(* CODESYS project RoboConnect_Dobot.library
   Company: RoboConnect
   DefaultNamespace: RoboConnect.Dobot
   Version: 0.1.0.0
   Placeholder: RoboConnect.Dobot
   Author: RoboConnect_Maintainers
   Description: 0.1.0.0 Branding update
      
      0.0.11.0 corrected MovJ arrays with checks
      0.0.10.0 adds free all tasks
      0.0.9.x - WIP
      0.0.9.0 refactors command creator
      0.0.8.0 updates to new Param name in TcRobot lib
      0.0.7.0 using new command infrastructure 
      0.0.0.6 command task receives 
      0.0.0.5 - updating array sizes
      0.0.0.3 adding receive packet scanning.
      0.0.0.2  adding separate port classes.
      0.0.0.1 Initial
   Title: RoboConnect.Dobot

Project tree, tasks and I/O mapping:
  libraries: Intecre.Utilities, * (Intecre Ltd); RoboConnect, * (RoboConnect); Tc2_Standard, * (Beckhoff Automation GmbH); Tc2_System, * (Beckhoff Automation GmbH); Tc2_Utilities, * (Beckhoff Automation GmbH)
  Commands and tasks/
    function block T_BoolCommandTaskV3 [ST]: Result, SetResultValue
    function block T_CommandTaskPoolV3 [ST]: FreeAllTasks, GetTask
    function block T_CommandTaskV3 [ST]: Abort, CyclicLogic, Execute, Free, Initalise, StateChanged, Available, Busy, Done, Error, ErrorId, Timeout
    function block T_DobotCommandConstructor [ST]: BrakeControl, ClearError, ContinueImmediate, ContinueScript, DisableRobot, EmergencyStop, EnableRobot, EnableRobotSpecifyCoG, Pause, PauseScript, PowerOn, ResetRobot, RunScript, SetCollideDrag, SetSafeSkin, StartDrag, StopDrag, StopScript, Wait, AccJ, AccL, CalcTool, CalcUser, Cp, LoadSwitch, PayLoad, SetArmOrientation, SetCollisionLevel, SetTool, SetUser, SpeedFactor, SpeedJ, SpeedL, TcpSpeed, TcpSpeedEnd, Tool, User, GetAngle, GetErrorID, GetPalletPose, GetPathStartPose, GetPose, GetSixForceData, GetTraceStartPose, HandleTrajPoints, InverseSolution, PalletCreate, PositiveSolution, RobotMode, AnalogueInput, AnalogueOutput, AoExecute, DigitalInput, DigitalOutput, DiGroup, DoExecute, DoGroup, GetTerminal485, SetTerminal485, ToolAI, ToolDI, ToolDO, ToolDOExecute, GetCoils, GetHoldRegs, GetInBits, GetInRegs, ModbusClose, ModbusCreate, SetCoils, SetHoldRegs, Circle3, Circle3Advanced, MoveJogCartesian, MoveJogCartesianAdvanced, MoveJogJointAxis, MoveJogJointAxisAdvanced, JointMovJ, JointMovJAdvanced, MovJ, MovJAdvanced, MovJIO, MovJIOAdvanced, MovL, MovLAdvanced, MovLIO, MovLIOAdvanced, RelJointMovJ, RelJointMovJAdvanced, RelMovJTool, RelMovJToolAdvanced, RelMovJUser, RelMovJUserAdvanced, RelMovLTool, RelMovLToolAdvanced, RelMovLUser, RelMovLUserAdvanced, ServoJ, ServoJAdvanced, Arc, ServoP, StartPath, StartTrace, Sync, CreateCommand, CreateCommand_EightArgs, CreateCommand_ElevenArgs, CreateCommand_Fifteen_Args, CreateCommand_FiveArgs, CreateCommand_FourArgs, CreateCommand_NineArgs, CreateCommand_OneArg, CreateCommand_SevenArgs, CreateCommand_SixArgs, CreateCommand_TenArgs, CreateCommand_Thirteen_Args, CreateCommand_ThreeArgs, CreateCommand_TwoArgs, CreateCommandNoArgs, EncapsulateWithCurlyBrax
    function block T_NumberCommandTaskV3 [ST]: Result, SetResultValue
  Helpers/
    function arrayToString [ST]
    function ByteArrayAdvanceAndClearRemaining [ST]
    function F_GetNextSegmentAndRemove [ST]
    function F_RemoveAfterSemiColon [ST]
    function F_RemoveAllOfACharacterInPlace [ST]
  Project Information/
    function F_GetCompany [ST]
    function F_GetTitle [ST]
    function F_GetVersion [ST]
  Structs and Enums/
    data type Converter2Bytes
    data type Converter8Bytes
    data type DOBOT_CMD_STRING
    data type DobotCR3Feedback
    data type E_BrakeControlRequest
    data type E_DobotTypes
    data type RobotModeConverter
    data type RobotModes
    data type TargetJogCrNova
  V3_API/
    function block T_DashboardV3 [ST]: ClearError, Disable, Enable, Halt, Reset, Stop, SetAnalogOutput, SetBufferMode, SetCarteasianAcceleration, SetCartesianDynamics, SetCartesianSpeed, SetDigitalOutput, SetJointAcceleration, SetJointSpeed, SetToolAnalogOutput, SetToolDigitalOutput, SetToolFrame, SetTransitionMode, SetTransitionParameter, SetUserFrame, ClearQueue, Connect, Disconnect, FreeAllTasks, SetRobotType, CallRobotApi, CallRobotApi_NormalPriority, Connected, DobotType
    function block T_FeedbackV3 [ST]: ClearAccumulator, Connect, CyclicReadFeedback, Disconnect, AdvanceAccumulatorArray, DecodeFeedback, Connected, Error, ErrorID, RobotFdBack
    function block T_MotionV3 [ST]: ClearQueue, Connect, Disconnect, FreeAllTasks, JogCartesian, JogJointAxis, MoveAbs, MoveJ, SetRobotType, CallRobotApi, CallRobotApi_NormalPriority, Connected, DobotType
    function block T_V3CommandAndFeedbackBaseClass [ST]: StateChanged, Connected, DobotType, CallRobotApi, ClearQueue, Connect, Disconnect, FreeAllTasks, Initialise, SetRobotType
    global variables V3_Ports
  Version/
    global variables Global_Version
  function block T_DobotV3_Cr_Nova [ST]: GetAnalogOutput, GetAxisCurrents, GetAxisPositions, GetAxisTemperatures, GetDigitalOutput, GetToolAnalogOutput, GetToolDigitalOutput, ClearError, Connect, CyclicLogic, Disable, Disconnect, Enable, FreeAllTasks, GetJointPositions, Halt, IsAtCartesianPosition, IsAtJointPosition, JogAxis, JogAxisAdvanced, JogCartesian, JogJointAxis, MoveAbs, MoveJ, Reset, SetAtPosDeltas, StateChanged, Stop, CartesianPosition, Connected, Enabled, Error, ErrorID, Manufacturer, Model, Running, ToolPosition, SetAnalogOutput, SetBufferMode, SetCarteasianAcceleration, SetCartesianDynamics, SetCartesianSpeed, SetDigitalOutput, SetJointAcceleration, SetJointSpeed, SetToolAnalogOutput, SetToolDigitalOutput, SetToolFrame, SetTransitionMode, SetTransitionParameter, SetUserFrame, FB_init, SetConnectionProperties
*)

// Structs and Enums/Converter2Bytes
TYPE Converter2Bytes :
UNION
	arrBytesIn : ARRAY[0..1] OF BYTE;
	realOut : INT;
END_UNION
END_TYPE

// Structs and Enums/Converter8Bytes
TYPE Converter8Bytes :
UNION
	arrBytesIn : ARRAY[0..7] OF BYTE;
	wordOut : LWORD;
	realOut : LREAL;
END_UNION
END_TYPE

// Structs and Enums/DOBOT_CMD_STRING
TYPE DOBOT_CMD_STRING : STRING(255); END_TYPE

// Structs and Enums/DobotCR3Feedback
TYPE DobotCR3Feedback :
STRUCT
	MessageSize : Converter2Bytes;
	DigitalInputs : ARRAY[0..8] OF BOOL;
	DigitalOutputs : ARRAY[0..8]OF BOOL;
	RobotMode : RobotModeConverter;
	TimeStamp : Converter8Bytes;
	TestValue :  Converter8Bytes;
	SpeedScaling : Converter8Bytes;
	LinearMomentumNorm : Converter8Bytes;
	VMain : Converter8Bytes;
	VRobot : Converter8Bytes;
	IRobot : Converter8Bytes;
	ToolAcceleroMeter : ARRAY[0..2] OF Converter8Bytes;
	ElbowPosition 	: ARRAY[0..2] OF Converter8Bytes;
	ElbowVelocity 	: ARRAY[0..2] OF Converter8Bytes;
	QTarget : ARRAY[0..5] OF Converter8Bytes; 	
	QDTarget : ARRAY[0..5] OF Converter8Bytes; 	
	QDDTarget : ARRAY[0..5] OF Converter8Bytes; 	
	ITarget : ARRAY[0..5] OF Converter8Bytes;	
	MTarget : ARRAY[0..5] OF Converter8Bytes;	
	QActual : ARRAY[0..5] OF Converter8Bytes;	
	QDActual : ARRAY[0..5] OF Converter8Bytes;
	IActual : ARRAY[0..5] OF Converter8Bytes;
	ActualTCPForce : ARRAY[0..5] OF Converter8Bytes;
	ToolVectorActual  : ARRAY[0..5] OF Converter8Bytes;	
	TCPSpeedActual : ARRAY[0..5] OF Converter8Bytes; 	
	TCPForce : ARRAY[0..5] OF Converter8Bytes; 	
	ToolVectorTarget : ARRAY[0..5] OF Converter8Bytes; 	
	TCPSpeedTarget : ARRAY[0..5] OF Converter8Bytes; 	
	MotorTemperatures : ARRAY[0..5] OF Converter8Bytes; 	
	JointModes : ARRAY[0..5] OF Converter8Bytes; 
	VActual : ARRAY[0..5] OF Converter8Bytes; 	
	HandType : ARRAY[0..3] OF BYTE; 	
	User : BYTE; 	
	Tool: Converter2Bytes;  	
	RunQueuedCmd: BOOL;  	
	PauseCmdFlag : BOOL; 	
	VelocityRatio: REAL;  	
	AccelerationRatio : REAL; 	
	JerkRatio 	: REAL; 
	XYZVelocityRatio: REAL;  	
	RVelocityRatio: REAL;  
	XYZAccelerationRatio: REAL;  	
	RAccelerationRatio : REAL; 	
	XYZJerkRatio : REAL; 	
	RJerkRatio : REAL; 	
	BrakeStatus : BOOL; 	
	EnableStatus : BOOL; 	
	DragStatus : BOOL; 	
	RunningStatus : BOOL; 	
	ErrorStatus : BOOL; 	
	JogStatusCR 	: BOOL; 
	CRRobotType : INT; 	
	DragButtonSignal : BOOL; 	
	EnableButtonSignal : BOOL; 	
	RecordButtonSignal : BOOL; 
	ReappearButtonSignal : BOOL; 	
	JawButtonSignal  : BOOL; 	
	SixForceOnline : BOOL; 	
	MActual : ARRAY[0..5] OF Converter8Bytes; 	 
	Load : ARRAY[0..4] OF REAL;  	
	CenterX : Converter2Bytes; 	
	CenterY  : Converter2Bytes;	
	CenterZ  : Converter2Bytes;	
//	User  : ARRAY[0..5] OF Converter8Bytes; 	 	
	ToolCordinates  : ARRAY[0..5] OF Converter8Bytes; 	 	
	TraceIndex : Converter8Bytes; 	
	SixForceValue  : ARRAY[0..5] OF Converter8Bytes; 		
	TargetQuaternion  : ARRAY[0..3] OF Converter8Bytes; 		
	ActualQuaternion : ARRAY[0..3] OF Converter8Bytes; 	
END_STRUCT
END_TYPE

// Structs and Enums/E_BrakeControlRequest
{attribute 'qualified_only'}
{attribute 'strict'}
TYPE E_BrakeControlRequest :
(
	NONE,
  ON,
  OFF
);
END_TYPE

// Structs and Enums/E_DobotTypes
{attribute 'qualified_only'}
{attribute 'to_string'}
{attribute 'strict'}
TYPE
E_DobotTypes :
(
  NONE,
  CR3, // 6 dof
  CR5, // 6 dof
  CR7, // 6 dof
  CR10, // 6 dof
  CR12, // 6 dof
  CR16, // 6 dof
  NOVA_2, // 6 dof
  NOVA_5, // 6 dof
  MG400 // 4 dof
);
END_TYPE

// Structs and Enums/RobotModeConverter
TYPE RobotModeConverter :
UNION
	arrBytesIn : ARRAY[0..7] OF BYTE;
	robotMode : INT;
END_UNION
END_TYPE

// Structs and Enums/RobotModes
{attribute 'qualified_only'}
{attribute 'to_string'}
TYPE
RobotModes :
(
  Not_Connected := 0,
  Initialization := 1,
  Brake_Release := 2,
  Disable := 4,
  Enable := 5,
  Dragging_State := 6,
  Running_State := 7,
  Draggin_Recording := 8,
  Alarm_State := 9,
  Pause_State := 10,
  Jogging_State := 11
) INT;
END_TYPE

// Structs and Enums/TargetJogCrNova
TYPE TargetJogCrNova :
(
	StopJog := 0,
	x := 1,
	y := 2,
	z := 3,
	a := 4,
	b := 5,
	c := 6	
);
END_TYPE

// V3_API/V3_Ports
{attribute 'qualified_only'}
VAR_GLOBAL CONSTANT
  FEEDBACK : UINT := 30004;
  DASHBOARD : UINT := 29999;
  MOTION : UINT := 30003;
END_VAR

// Version/Global_Version
{attribute 'TcGenerated'}
{attribute 'no-analysis'}
{attribute 'linkalways'}
// This function has been automatically generated from the project information.
VAR_GLOBAL CONSTANT
	{attribute 'const_non_replaced'}
	stLibVersion_RoboConnect_Dobot : ST_LibVersion := (iMajor := 0, iMinor := 1, iBuild := 0, iRevision := 0, nFlags := 0, sVersion := '0.1.0.0');
END_VAR

// Commands and tasks/T_BoolCommandTaskV3
FUNCTION_BLOCK T_BoolCommandTaskV3 EXTENDS T_CommandTaskV3 IMPLEMENTS I_BoolResultTask
VAR
  _boolResult : BOOL;
END_VAR

PROPERTY Result : BOOL
GET
Result := _boolResult;
END_GET
END_PROPERTY

METHOD PUBLIC SetResultValue
VAR_INPUT
  value : BOOL;
END_VAR
_boolResult := value;
END_METHOD

END_FUNCTION_BLOCK

// Commands and tasks/T_CommandTaskV3
FUNCTION_BLOCK T_CommandTaskV3 EXTENDS T_NamedBase IMPLEMENTS I_CommandTask
VAR
  _busy : BOOL := FALSE;
  _error : BOOL := FALSE;
  _done : BOOL := FALSE;
  _errorId : STRING;
  _result : DOBOT_CMD_STRING;
  _timeout : BOOL := FALSE;
  _available : BOOL := TRUE;

  state, prevState : (UNINITLIASED,
    INITALISED,
    SENDING,
    WAITING_FOR_RESPONSE,
    DONE_STATE,
    ERROR_STATE);

  _comPort : I_Connection;
  _msg : T_Maxstring;
  
  timeoutTimer : TON := (PT := TASK_TIMEOUT);
  data : RecvBuffer;
  receiveLength : UDINT;
  resultString : DOBOT_CMD_STRING;
  origRequestPosition : INT;
  errorString : T_Maxstring;
  originalReq : DOBOT_CMD_STRING;
  errorCode : DOBOT_CMD_STRING;
  results : DOBOT_CMD_STRING;
  spaceString : STRING := ' ';
  tempResString : DOBOT_CMD_STRING;

END_VAR
VAR CONSTANT
  TASK_TIMEOUT : TIME := RoboConnect.RoboConnectParams.TimeOut;
END_VAR

METHOD Abort
END_METHOD

METHOD PUBLIC CyclicLogic
CASE state OF
  UNINITLIASED:
    StateChanged();

  INITALISED:
    IF StateChanged() THEN
      logInfo('task initlaised');
    END_IF

  SENDING:
    IF StateChanged() THEN
      _busy := TRUE;
      timeoutTimer.IN := FALSE;

      IF NOT _comPort.Send(_msg) THEN
        state := ERROR_STATE;
        RETURN;

      END_IF

    ELSE
      timeoutTimer.IN := TRUE;
    END_IF

    IF timeoutTimer.Q THEN
      state := ERROR_STATE;
      LogError('Command timed out');
    END_IF

    IF _comPort.SendDone THEN
      state := WAITING_FOR_RESPONSE;
    END_IF

  WAITING_FOR_RESPONSE:
    timeoutTimer.IN := NOT StateChanged();

    IF timeoutTimer.Q THEN
      LogError('No return from sent command!');
      state := ERROR_STATE;

    ELSIF _comPort.IsErrorConnect OR _comPort.IsErrorReceive THEN
      LogError('_comPort.IsErrorConnect OR _comPort.IsErrorReceive');
      state := ERROR_STATE;

    ELSIF _comPort.Receive(data => data, receiveLength => receiveLength) THEN
      // convert to string
      MEMCPY(ADR(resultString), ADR(data), receiveLength);

      // Break up parts of the command
      errorCode := F_GetNextSegmentAndRemove(resultString, ',');
      results := F_GetNextSegmentAndRemove(resultString, ',');
      originalReq := F_RemoveAfterSemiColon(resultString);
      F_RemoveAllOfACharacterInPlace(original := originalReq, stringToRemove := spaceString );

      // Check what was send is what was received 
      IF originalReq = _msg THEN
        _errorId := errorCode;
        _error := errorCode <> TO_STRING(0);
        _result := results;
        state := DONE_STATE;

      ELSE
        LogError(CONCAT('Response does not contain request:', originalReq));
        LogError(CONCAT('Original request:', _msg));
        state := ERROR_STATE;

      END_IF
    END_IF

  DONE_STATE:
    IF StateChanged() THEN
      LogInfo('task done');
      _busy := FALSE;
      _done := TRUE;
      timeoutTimer.IN := FALSE;
    END_IF

  ERROR_STATE:
    IF StateChanged() THEN
      LogError('task error');
      _error := TRUE;
      _busy := FALSE;
      _done := FALSE;
    END_IF

END_CASE

timeoutTimer();
END_METHOD

METHOD PUBLIC Execute : BOOL
IF state <> INITALISED THEN
  RETURN;
END_IF

state := SENDING;
Execute := TRUE;
END_METHOD

METHOD PUBLIC Free
_Busy := FALSE;
_Error := FALSE;
_Done := FALSE;
 _timeout := FALSE;
 _available := TRUE;
  
_comPort := 0;
_msg := '';
END_METHOD

METHOD PUBLIC Initalise : BOOL
VAR_INPUT
 comPort : I_Connection;
 msg : T_Maxstring;
END_VAR
IF comPort = 0 THEN
  RETURN;
END_IF

_done := FALSE;
_comPort := comPort;
_msg := msg;
state := INITALISED;
Initalise := TRUE;
_available := false;
END_METHOD

METHOD PRIVATE StateChanged : BOOL
IF  state = prevState THEN
  RETURN;
END_IF

prevState := state;
StateChanged := TRUE;
END_METHOD

PROPERTY Available : BOOL
GET
Available := _available;
END_GET
END_PROPERTY

PROPERTY Busy : BOOL
GET
Busy := _Busy;
END_GET
END_PROPERTY

PROPERTY Done : BOOL
GET
Done := _Done;
END_GET
END_PROPERTY

PROPERTY Error : BOOL
GET
Error := _error;
END_GET
END_PROPERTY

PROPERTY PUBLIC ErrorId : STRING
GET
ErrorId := _errorId;
END_GET
END_PROPERTY

PROPERTY Timeout : BOOL
GET
Timeout := _timeout;
END_GET
END_PROPERTY

END_FUNCTION_BLOCK

// Helpers/F_GetNextSegmentAndRemove
FUNCTION INTERNAL F_GetNextSegmentAndRemove : STRING // returned segment. Does not include split character
VAR_IN_OUT
	OriginalString : STRING; // this string will be modified if split character found.
END_VAR
VAR_INPUT
	CharacterToSplitOn : STRING; // first character of this string shall be used	
END_VAR

IF LEN( OriginalString ) > 0 AND_THEN LEN( CharacterToSplitOn ) > 0 THEN

	F_GetNextSegmentAndRemove := 
		LEFT( 
			OriginalString, 
			FIND( OriginalString, LEFT( CharacterToSplitOn, 1 ) ) - 1 // do not retun the splitting character
		);
		
	OriginalString := 
		DELETE(
			OriginalString, 
			FIND( OriginalString, LEFT( CharacterToSplitOn, 1 ) ), 
			1 
		);
		
END_IF

END_FUNCTION

// Helpers/F_RemoveAfterSemiColon
FUNCTION F_RemoveAfterSemiColon : STRING
VAR_IN_OUT
  OriginalString : STRING;
END_VAR
VAR
  semiColonIndex : INT;
  semiColon : STRING := ';';
END_VAR

IF LEN(OriginalString) > 1 THEN
  semiColonIndex := FIND(OriginalString, semiColon);
  OriginalString := LEFT(OriginalString, semiColonIndex - 1);
  F_RemoveAfterSemiColon := LEFT(OriginalString, semiColonIndex - 1);
END_IF

END_FUNCTION

// Helpers/F_RemoveAllOfACharacterInPlace
FUNCTION F_RemoveAllOfACharacterInPlace 
VAR_IN_OUT
  original : DOBOT_CMD_STRING;
END_VAR
VAR_INPUT
  stringToRemove : STRING;
END_VAR
VAR
  _stringToRemove : STRING := ' ';
  tempResString : DOBOT_CMD_STRING;
END_VAR

_stringToRemove := stringToRemove;

WHILE FindAndDelete(
  pSrcString := ADR(original),
  pDeleteString := ADR(_stringToRemove),
  pDstString := ADR(tempResString),
  nDstSize := SIZEOF(tempResString)
      )
        > 0 DO

  // put back in to recursively remove spaces
  original := tempResString;

END_WHILE

END_FUNCTION

// Commands and tasks/T_CommandTaskPoolV3
FUNCTION_BLOCK T_CommandTaskPoolV3 IMPLEMENTS I_TaskPool
VAR
  taskList : ARRAY [0..MAX_TASK_SIZE] OF T_CommandTaskV3;
END_VAR
VAR CONSTANT
  MAX_TASK_SIZE : UINT := 56;
END_VAR

METHOD PUBLIC FreeAllTasks
VAR
  i : UINT;
END_VAR
FOR i := 0 TO MAX_TASK_SIZE DO
  taskList[i].Free();
END_FOR
END_METHOD

METHOD PUBLIC GetTask : BOOL
VAR_OUTPUT
  result : I_CommandTask;
END_VAR
VAR
  i : UINT;
END_VAR
FOR i := 0 TO MAX_TASK_SIZE DO
  IF taskList[i].Available THEN
    result := taskList[i];
    GetTask := TRUE;
    RETURN;
  END_IF
END_FOR

GetTask := FALSE;
END_METHOD

END_FUNCTION_BLOCK

// Commands and tasks/T_DobotCommandConstructor
FUNCTION_BLOCK T_DobotCommandConstructor EXTENDS T_NamedBase

METHOD BrakeControl : BOOL
VAR_INPUT
	axisID : INT; //joint ID, 1: J1, 2: J2, and so on
	brakeRequest : E_BrakeControlRequest; 
END_VAR
VAR_OUTPUT
	commandOutput : DOBOT_CMD_STRING;
END_VAR
VAR
  translatedBrakeValue : INT; // from Doboot API 0: Switch off brake, 1: Switch on brake
END_VAR
VAR CONSTANT
  BRAKE_CONTROL_CMD : STRING := 'BrakeControl';
END_VAR
CASE brakeRequest OF

  E_BrakeControlRequest.ON:
    translatedBrakeValue := 1;

  E_BrakeControlRequest.OFF:
    translatedBrakeValue := 0;

ELSE

  LogWarning('Cannot request Brake Control as brakeRequest = E_BrakeControlRequest.NONE ');
  RETURN;

END_CASE

commandOutput := CreateCommand_TwoArgs(BRAKE_CONTROL_CMD, TO_STRING(axisID), TO_STRING(translatedBrakeValue));

BrakeControl := TRUE;
END_METHOD

METHOD ClearError : BOOL
VAR_OUTPUT
	commandOutput : DOBOT_CMD_STRING;
END_VAR
VAR CONSTANT
	CLEAR_ERROR_CMD : STRING := 'ClearError';
END_VAR
commandOutput := CreateCommandNoArgs(CLEAR_ERROR_CMD);
ClearError := TRUE;
END_METHOD

METHOD ContinueImmediate : BOOL
VAR_OUTPUT
	commandOutput : DOBOT_CMD_STRING;
END_VAR
VAR CONSTANT
	CONTINUE_IMMEDIATE_CMD : STRING := 'Continue';
END_VAR
commandOutput := CreateCommandNoArgs(CONTINUE_IMMEDIATE_CMD);
ContinueImmediate := TRUE;
END_METHOD

METHOD ContinueScript : BOOL
VAR_OUTPUT
	commandOutput : DOBOT_CMD_STRING;
END_VAR
VAR CONSTANT
	CONTINUE_SCRIPT_CMD : STRING := 'ContinueScript';
END_VAR
commandOutput := CreateCommandNoArgs(CONTINUE_SCRIPT_CMD);
ContinueScript := TRUE;
END_METHOD

METHOD DisableRobot : BOOL
VAR_OUTPUT
	commandOutput : DOBOT_CMD_STRING;
END_VAR
VAR CONSTANT
	DISABLE_ROBOT_CMD : STRING := 'DisableRobot';
END_VAR
commandOutput := CreateCommandNoArgs(DISABLE_ROBOT_CMD);
DisableRobot := TRUE;
END_METHOD

METHOD EmergencyStop : BOOL
VAR_OUTPUT
	commandOutput : DOBOT_CMD_STRING;
END_VAR
VAR CONSTANT
	EMERGENCY_STOP_CMD : STRING := 'EmergencyStop';
END_VAR
commandOutput := CreateCommandNoArgs(EMERGENCY_STOP_CMD);
EmergencyStop := TRUE;
END_METHOD

METHOD EnableRobot : BOOL
VAR_OUTPUT
	commandOutput : DOBOT_CMD_STRING;
END_VAR
VAR CONSTANT
	ENABLE_ROBOT_CMD : DOBOT_CMD_STRING := 'EnableRobot';
END_VAR
commandOutput := CreateCommandNoArgs(ENABLE_ROBOT_CMD);
EnableRobot := TRUE;
END_METHOD

METHOD EnableRobotSpecifyCoG : BOOL // enable while specifying load and load CoG.
{attribute 'obsolete' := 'This input is optional'}
VAR_INPUT
  load : REAL := 0; //Load weight.The value range should not exceed the load range of corresponding robot models, unit: kg.
  centreX : REAL := 0; //Eccentric distance in X-axis direction. Range: -500 – 500, unit: mm.
  centreY : REAL := 0; //Eccentric distance in Y-axis direction. Range: -500 – 500, unit: mm.
  centreZ : REAL := 0; //Eccentric distance in Z-axis direction. Range: -500 – 500, unit: mm.
END_VAR
VAR_OUTPUT
  commandOutput : DOBOT_CMD_STRING;
END_VAR
VAR CONSTANT
  UPPER_LOAD_DISTANCE_BOUND : LREAL := 500; // mm
  LOWER_LOAD_DISTANCE_BOUND : LREAL := -500; // mm
  ENABLE_ROBOT_CMD : STRING := 'EnableRobot';
END_VAR
IF centreX < LOWER_LOAD_DISTANCE_BOUND OR centreX > UPPER_LOAD_DISTANCE_BOUND THEN
  LogWarning(
    CONCAT('cannot EnableRobotSpecifyCoG as centerX exceeds bounds : ', TO_STRING(centreX))
  );

  RETURN;

END_IF

IF centreY < LOWER_LOAD_DISTANCE_BOUND OR centreY > UPPER_LOAD_DISTANCE_BOUND THEN
  LogWarning(
    CONCAT('cannot EnableRobotSpecifyCoG as centreY exceeds bounds : ', TO_STRING(centreY))
  );

  RETURN;

END_IF

IF centreZ < LOWER_LOAD_DISTANCE_BOUND OR centreZ > UPPER_LOAD_DISTANCE_BOUND THEN
  LogWarning(
    CONCAT('cannot EnableRobotSpecifyCoG as centreZ exceeds bounds : ', TO_STRING(centreZ))
  );

  RETURN;

END_IF

commandOutput := CreateCommand_FourArgs(
  ENABLE_ROBOT_CMD,
  TO_STRING(load),
  TO_STRING(centreX),
  TO_STRING(centreY),
  TO_STRING(centreZ)
);

EnableRobotSpecifyCoG := TRUE;
END_METHOD

METHOD Pause : BOOL
VAR_OUTPUT
	commandOutput : DOBOT_CMD_STRING;
END_VAR
VAR CONSTANT
	PAUSE_CMD : STRING := 'Pause';
END_VAR
commandOutput := CreateCommandNoArgs(PAUSE_CMD);
Pause := TRUE;
END_METHOD

METHOD PauseScript : BOOL
VAR_OUTPUT
	commandOutput : DOBOT_CMD_STRING;
END_VAR
VAR CONSTANT
	PAUSE_SCRIPT_CMD : STRING := 'PauseScript';
END_VAR
commandOutput := CreateCommandNoArgs(PAUSE_SCRIPT_CMD);
PauseScript := TRUE;
END_METHOD

METHOD PowerOn : BOOL 
VAR_OUTPUT
	commandOutput : STRING;
END_VAR
VAR
	POWER_ON_CMD : STRING := 'PowerOn';
END_VAR
commandOutput := CreateCommandNoArgs(POWER_ON_CMD);
PowerOn := TRUE;
END_METHOD

METHOD ResetRobot : BOOL
VAR_OUTPUT
	commandOutput : DOBOT_CMD_STRING;
END_VAR
VAR CONSTANT
	RESET_ROBOT_CMD : STRING := 'ResetRobot';
END_VAR
commandOutput := CreateCommandNoArgs(RESET_ROBOT_CMD);
ResetRobot := TRUE;
END_METHOD

METHOD RunScript : BOOL
VAR_INPUT
	projectName : STRING; //Project name as created using Dobot Studio Pro
END_VAR
VAR_OUTPUT
	commandOutput : DOBOT_CMD_STRING;
END_VAR
VAR CONSTANT
	RUN_SCRIPT_CMD : STRING := 'RunScript';
END_VAR
commandOutput := CreateCommand_OneArg(RUN_SCRIPT_CMD, projectName);
RunScript := TRUE;
END_METHOD

METHOD SetCollideDrag : BOOL
VAR_INPUT
	status : INT; //Forced drag switch. 0: Forced to exit the drag mode. 1: forced to enter the drag mode.
END_VAR
VAR_OUTPUT
	commandOutput : DOBOT_CMD_STRING;
END_VAR
VAR CONSTANT
	SET_COLLIDE_DRAG_CMD : STRING := 'SetCollideDrag';
END_VAR
commandOutput := CreateCommand_OneArg(baseCommand := SET_COLLIDE_DRAG_CMD, arg_01 := TO_STRING(status));

SetCollideDrag := TRUE;
END_METHOD

METHOD SetSafeSkin : BOOL
VAR_INPUT
  status : INT; //SafeSkin switch, 0: off, 1: on
END_VAR
VAR_OUTPUT
  commandOutput : DOBOT_CMD_STRING;
END_VAR
VAR CONSTANT
  SET_SAFE_SKIN_CMD : STRING := 'SetSafeSkin';
END_VAR
commandOutput := CreateCommand_OneArg(baseCommand := SET_SAFE_SKIN_CMD, arg_01 := TO_STRING(status));

setSafeSkin := TRUE;
END_METHOD

METHOD StartDrag : BOOL
VAR_OUTPUT
	commandOutput : DOBOT_CMD_STRING;
END_VAR
VAR CONSTANT
	START_DRAG_CMD : STRING := 'StartDrag';
END_VAR
commandOutput := CreateCommandNoArgs( START_DRAG_CMD);
startDrag := TRUE;
END_METHOD

METHOD StopDrag : BOOL
VAR_OUTPUT
	commandOutput : DOBOT_CMD_STRING;
END_VAR
VAR CONSTANT
	STOP_DRAG_CMD : STRING := 'StopDrag';
END_VAR
commandOutput := CreateCommandNoArgs(STOP_DRAG_CMD);
stopDrag := TRUE;
END_METHOD

METHOD StopScript : BOOL
VAR_OUTPUT
	commandOutput : DOBOT_CMD_STRING;
END_VAR
VAR CONSTANT
	STOP_SCRIPT_CMD : DOBOT_CMD_STRING := 'StopScript';
END_VAR
commandOutput := CreateCommandNoArgs( STOP_SCRIPT_CMD);
stopScript := TRUE;
END_METHOD

METHOD Wait : BOOL
VAR_INPUT
  timeToWait : INT; //Delayed time, unit:ms, range: (0,3600*1000)
END_VAR
VAR_OUTPUT
  commandOutput : DOBOT_CMD_STRING;
END_VAR
VAR CONSTANT
  WAIT_CMD : STRING := 'Wait';
END_VAR
commandOutput := CreateCommand_OneArg(baseCommand := WAIT_CMD, arg_01 := TO_STRING(timeToWait));

Wait := TRUE;
END_METHOD

METHOD AccJ : BOOL
VAR_INPUT
	acc : INT ; //Acceleration ratio: [1-100]
END_VAR
VAR_OUTPUT
	commandOutput : DOBOT_CMD_STRING;
END_VAR
VAR CONSTANT
	ACC_J_CMD : STRING := 'AccJ';
END_VAR
commandOutput := CreateCommand_OneArg(baseCommand := ACC_J_CMD, arg_01 := TO_STRING(acc));
AccJ := TRUE;
END_METHOD

METHOD AccL : BOOL
VAR_INPUT
	acc : INT ; //Acceleration ratio: [1-100]
END_VAR
VAR_OUTPUT
	commandOutput : DOBOT_CMD_STRING;
END_VAR
VAR CONSTANT
	ACC_L_CMD : STRING := 'AccL';
END_VAR
commandOutput := CreateCommand_OneArg(baseCommand := ACC_L_CMD, arg_01 := TO_STRING(acc) );
accL := TRUE;
END_METHOD

METHOD CalcTool : BOOL
VAR_INPUT
	index : INT ; //Index of the user coordinate system, range: [0,9]. The initial value of coordinate system 0 is the base coordinate system.
	matrix_direction : INT; //Calculation method. 1: left multiplication, indicating that the coordinate system specified by "index" deflects the value specified by "table" along the flange coordinate system. 0: right multiplication, indicating that the coordinate system specified by "index" deflects the value specified by "table" along itself.
	table : STRING; //User coordinate system offset, format :{x, y, z, rx, ry, rz}.
END_VAR
VAR_OUTPUT
	commandOutput : DOBOT_CMD_STRING;
END_VAR
VAR CONSTANT
	CALC_TOOL_CMD : STRING := 'CalcTool';
END_VAR
commandOutput := CreateCommand_ThreeArgs(
  baseCommand := CALC_TOOL_CMD,
  TO_STRING(index),
  TO_STRING(matrix_direction),
  EncapsulateWithCurlyBrax(table)
);

calcTool := TRUE;
END_METHOD

METHOD CalcUser : BOOL
VAR_INPUT
	index : INT; //Index of the user coordinate system, range: [0,9]. The initial value of coordinate system 0 is the base coordinate system.
	matrix_direction : INT; //Calculation method. 1: left multiplication, indicating that the coordinate system specified BY "index" deflects the value specified BY "table" along the base coordinate system. 0: right multiplication, indicating that the coordinate system specified by "index" deflects the value specified by "table" along itself.
	table : STRING; //User coordinate system offset, format :{x, y, z, rx, ry, rz}.
END_VAR
VAR_OUTPUT
	commandOutput : DOBOT_CMD_STRING;
END_VAR
VAR CONSTANT
	CALC_USER_CMD : STRING := 'CalcUser';
END_VAR
commandOutput := CreateCommand_ThreeArgs(
  baseCommand := CALC_USER_CMD,
  TO_STRING(index),
  TO_STRING(matrix_direction),
  EncapsulateWithCurlyBrax(table)
);

calcUser := TRUE;
END_METHOD

METHOD Cp : BOOL
VAR_INPUT
	ratio : LREAL ; //Continuous path ratio: [1-100]
END_VAR
VAR_OUTPUT
	commandOutput : DOBOT_CMD_STRING;
END_VAR
VAR CONSTANT
	CP_CMD : STRING := 'CP';
END_VAR
commandOutput := CreateCommand_OneArg(baseCommand := CP_CMD, arg_01 := TO_STRING(ratio));
Cp := TRUE;
END_METHOD

METHOD LoadSwitch : BOOL
VAR_INPUT
	status : INT ; //Load setting switch. 0: off, 1: on
END_VAR
VAR_OUTPUT
	commandOutput : DOBOT_CMD_STRING;
END_VAR
VAR CONSTANT
	LOAD_SWITCH_CMD : STRING := 'LoadSwitch';
END_VAR
commandOutput := CreateCommand_OneArg(LOAD_SWITCH_CMD, TO_STRING(status));
LoadSwitch := TRUE;
END_METHOD

METHOD PayLoad : BOOL
VAR_INPUT
	weight : REAL; //Load weight. The value range should not exceed the load range of the corresponding robot model. unit kg
	interia : REAL; //Load inertia. unit kgm^2
END_VAR
VAR_OUTPUT
	commandOutput : DOBOT_CMD_STRING;
END_VAR
VAR
	PAY_LOAD_CMD : STRING := 'PayLoad';
END_VAR
commandOutput := CreateCommand_TwoArgs(PAY_LOAD_CMD, TO_STRING(weight), TO_STRING(interia));
PayLoad := TRUE;
END_METHOD

METHOD SetArmOrientation : BOOL
VAR_INPUT
	lorr : INT ; //Orientation of the upper arm. 1: forward (joint angle of J2: positive), -1: backward (joint angle of J2: negative).
	uord : INT; //Orientation of the elbow joint. 1: upward (joint angle of J3: positive), -1: downward (joint angle of J3: negative).
	forn : INT; //Indicates whether the wrist joint is flipped or not. 1: wrist joint is not flipped (joint angle of J5: positive), -1: wrist joint is flipped (joint angle of J5: negative).
	config6 : INT; //J6 angle range.-1: [0, -90], -2: [-90, -180], 1: [0, 90], 2: [90, 180] ...
END_VAR
VAR_OUTPUT
	commandOutput : DOBOT_CMD_STRING;
END_VAR
VAR CONSTANT
	commandBase : STRING := 'SetArmOrientation';
END_VAR
commandOutput := CreateCommand_FourArgs(
  commandBase,
  TO_STRING(lorr),
  TO_STRING(uord),
  TO_STRING(forn),
  TO_STRING(config6)
);

SetArmOrientation := TRUE;
END_METHOD

METHOD SetCollisionLevel : BOOL
VAR_INPUT
	level : INT ; //Collision detection level. 0: switching off collision detection. 1 – 5: the larger the number, the higher the sensitivity.
END_VAR
VAR_OUTPUT
	commandOutput : DOBOT_CMD_STRING;
END_VAR
VAR CONSTANT
	SET_COLLISION_LEVEL_CMD : STRING := 'SetCollisionLevel';
END_VAR
IF level < 0 OR level > 5 THEN
  LogError(
    CONCAT(
      'Invalid collision level: ',
      TO_STRING(level)
    )
  );
  RETURN;
  
END_IF

commandOutput := CreateCommand_OneArg(SET_COLLISION_LEVEL_CMD, TO_STRING(level));
SetCollisionLevel := TRUE;
END_METHOD

METHOD SetTool : BOOL
VAR_INPUT
	index : INT; //Index of the tool coordinate system, range: [0,9]. The initial value of coordinate system 0 is the flange coordinate system.
	table : STRING; //Tool coordinate system after modification, format: {x, y, z, rx, ry, rz}, which is recommended to obtain through CalcTool command
END_VAR
VAR_OUTPUT
	commandOutput : DOBOT_CMD_STRING;
END_VAR
VAR CONSTANT
	SET_TOOL_CMD : STRING := 'SetTool';
END_VAR
commandOutput := CreateCommand_TwoArgs(
  SET_TOOL_CMD,
  TO_STRING(index),
  EncapsulateWithCurlyBrax(table)
);

SetTool := TRUE;
END_METHOD

METHOD SetUser : BOOL
VAR_INPUT
	index : INT ; //Index of the user coordinate system, range :[0,9]. The initial value of coordinate system 0 is the base coordinate system.
	table : STRING ; // User coordinate system after modification, format:{x,y,z,rx,ry,rz}, which is recommended to obtain through CalcUser command.
END_VAR
VAR_OUTPUT
	commandOutput : DOBOT_CMD_STRING;
END_VAR
VAR CONSTANT
	SET_USER_CMD : STRING := 'SetUser';
END_VAR
commandOutput := CreateCommand_TwoArgs(
  SET_USER_CMD,
  TO_STRING(index),
  EncapsulateWithCurlyBrax(table)
);

SetUser := TRUE;
END_METHOD

METHOD SpeedFactor : BOOL
VAR_INPUT
	ratio : INT ; //DGlobal speed ratio, range 1-100
END_VAR
VAR_OUTPUT
	commandOutput : DOBOT_CMD_STRING;
END_VAR
VAR CONSTANT
	SPEED_FACTOR_CMD : STRING := 'SpeedFactor';
END_VAR
commandOutput := CreateCommand_OneArg(SPEED_FACTOR_CMD, TO_STRING(ratio));
SpeedFactor := TRUE;
END_METHOD

METHOD SpeedJ : BOOL
VAR_INPUT
	speed : INT ; //Speed ratio: [1-100]
END_VAR
VAR_OUTPUT
	commandOutput : DOBOT_CMD_STRING;
END_VAR
VAR CONSTANT
	SPEED_J_CMD : STRING := 'SpeedJ';
END_VAR
commandOutput := CreateCommand_OneArg(SPEED_J_CMD, TO_STRING(speed));
SpeedJ := TRUE;
END_METHOD

METHOD SpeedL : BOOL
VAR_INPUT
	speed : INT ; //Speed ratio: [1-100]
END_VAR
VAR_OUTPUT
	commandOutput : DOBOT_CMD_STRING;
END_VAR
VAR CONSTANT
	SPEED_L_CMD : STRING := 'SpeedL';
END_VAR
commandOutput := CreateCommand_OneArg(SPEED_L_CMD, TO_STRING(speed));
SpeedL := TRUE;
END_METHOD

METHOD TcpSpeed : BOOL
VAR_INPUT
	vt : USINT; //Absolute speed, unit: mm/s, range: [0,100000]
END_VAR
VAR_OUTPUT
	commandOutput : DOBOT_CMD_STRING;
END_VAR
VAR CONSTANT
	TCP_SPEED_CMD : STRING := 'TCPSpeed';
END_VAR
commandOutput := CreateCommand_OneArg(TCP_SPEED_CMD, TO_STRING(VT));
TcpSpeed := TRUE;
END_METHOD

METHOD TcpSpeedEnd : BOOL
VAR_OUTPUT
	commandOutput : DOBOT_CMD_STRING;
END_VAR
VAR CONSTANT
	TCP_SPEED_END_CMD : STRING := 'TCPSpeedEnd';
END_VAR
commandOutput := CreateCommandNoArgs(baseCommand := TCP_SPEED_END_CMD);
TcpSpeedEnd := TRUE;
END_METHOD

METHOD Tool : BOOL
VAR_INPUT
	status : INT ; //Load settign switch 0: off, 1:on 
END_VAR
VAR_OUTPUT
	commandOutput : STRING;
END_VAR
VAR CONSTANT
	TOOL_CMD : STRING := 'Tool';
END_VAR
commandOutput := 
  CreateCommand_OneArg(TOOL_CMD, TO_STRING(status));
Tool := TRUE;
END_METHOD

METHOD User : BOOL
VAR_INPUT
	index : INT ; //Index of the calibrated user coordinate system, which needs to be calibrated by software before it can be selected here. 
END_VAR
VAR_OUTPUT
	commandOutput : DOBOT_CMD_STRING;
END_VAR
VAR
	USER_CMD : STRING := 'User';
END_VAR
commandOutput := CreateCommand_OneArg(USER_CMD, TO_STRING(index));
User := TRUE;
END_METHOD

METHOD GetAngle : BOOL
VAR_OUTPUT
	commandOutput : DOBOT_CMD_STRING;
END_VAR
VAR
	GET_ANGLE_CMD : STRING := 'GetAngle';
END_VAR
commandOutput := GET_ANGLE_CMD;
GetAngle := TRUE;
RETURN;
END_METHOD

METHOD GetErrorID : BOOL
VAR_OUTPUT
	commandOutput : DOBOT_CMD_STRING;
END_VAR
VAR
	GET_ERROR_ID_CMD : STRING := 'GetErrorID';
END_VAR
commandOutput := GET_ERROR_ID_CMD;
getErrorID := TRUE;
RETURN;
END_METHOD

METHOD GetPalletPose : BOOL
VAR_INPUT
	palletName : STRING ; //Pallet name
	index : INT; //Point index, starting from 1
END_VAR
VAR_OUTPUT
	commandOutput : DOBOT_CMD_STRING;
END_VAR
VAR
	GET_PALLET_POSE_CMD : STRING := 'GetPalletPose';
END_VAR
commandOutput := CreateCommand_TwoArgs(GET_PALLET_POSE_CMD, palletName, TO_STRING(index));
GetPalletPose := TRUE;
END_METHOD

METHOD GetPathStartPose : BOOL
VAR_INPUT
	traceName : STRING ; //Trajectory file name (with suffix) The trajectory file is stored in /dobot/userdata/project/process/trajectory/.
END_VAR
VAR_OUTPUT
	commandOutput : DOBOT_CMD_STRING;
END_VAR
VAR CONSTANT
	GET_PATH_START_POSE_CMD : STRING := 'GetPathStartPose';
END_VAR
commandOutput := CreateCommand_OneArg(GET_PATH_START_POSE_CMD,traceName);
GetPathStartPose := TRUE;
END_METHOD

METHOD GetPose : BOOL
VAR_INPUT
	user : INT ; //Index of the calibrated user coordinate system
	tool : INT; //Index of the calibrated tool coordinate system
END_VAR
VAR_OUTPUT
	commandOutput : STRING;
END_VAR
VAR CONSTANT 
  	GET_POSE_CMD : STRING := 'GetPose';
END_VAR
commandOutput := CreateCommand_TwoArgs(GET_POSE_CMD, TO_STRING(user), TO_STRING(tool));
GetPose := TRUE;
END_METHOD

METHOD GetSixForceData : BOOL
VAR_OUTPUT
	commandOutput : DOBOT_CMD_STRING;
END_VAR
VAR CONSTANT
  	GET_SIX_FORCE_DELTA_CMD : STRING := 'GetSixForceData';
END_VAR
commandOutput := CreateCommandNoArgs(GET_SIX_FORCE_DELTA_CMD);
GetSixForceData := TRUE;
END_METHOD

METHOD GetTraceStartPose : BOOL
VAR_INPUT
	traceName : STRING ; //trajectory file name (with suffix) The trajectory file is stored in /dobot/userdata/project/process/trajectory/.
END_VAR
VAR_OUTPUT
	commandOutput : DOBOT_CMD_STRING;
END_VAR
VAR CONSTANT
  GET_TRACE_START_POSE_CMD : STRING := 'GetTraceStartPose';
END_VAR
commandOutput := CreateCommand_OneArg(GET_TRACE_START_POSE_CMD, traceName);
GetTraceStartPose := TRUE;
END_METHOD

METHOD HandleTrajPoints : BOOL
VAR_INPUT
	traceName : STRING ; //trajectory file name (with suffix) The trajectory file is stored in /dobot/userdata/project/process/trajectory/.
END_VAR
VAR_OUTPUT
	commandOutput : DOBOT_CMD_STRING;
END_VAR
VAR CONSTANT
  HANDLE_TRAJ_POINTS_CMD : STRING := 'HandleTrajPoints';
END_VAR
commandOutput := CreateCommand_OneArg(HANDLE_TRAJ_POINTS_CMD, traceName);
HandleTrajPoints := TRUE;
END_METHOD

METHOD InverseSolution : BOOL
VAR_INPUT
	x : REAL ; //X-axis position, unit: mm
	y : REAL ; //Y-axis position, unit: mm
	z : REAL ; //Z-axis position, unit: mm
	rX : REAL; //Rx-axis position, unit: °
	rY : REAL; //Ry-axis position, unit: °
	rZ : REAL; //Rz-axis position, unit: °
	user : INT; //Index of the calibrated user coordinate system
	tool : INT; //Index of the calibrated tool coordinate system
	isJointNear : INT; //Optional parameter. It is used to set whether JointNear is effective. If the value is 0 or null, JointNear data is ineffective. The algorithm selects the joint angles according to the current angle. If the value is 1, the algorithm selects the joint angles according to JointNear data.
	jointNear : INT; //Optional parameter. Joint coordinates for selecting joint angles. 
END_VAR
VAR_OUTPUT
	commandOutput : DOBOT_CMD_STRING;
END_VAR
VAR CONSTANT
  INVERSE_SOLUTION_CMD : STRING := 'InverseSolution';
END_VAR
IF isJointNear = 0 AND jointNear = 0 THEN
  commandOutput := CreateCommand_EightArgs(
    INVERSE_SOLUTION_CMD,
    TO_STRING(x),
    TO_STRING(y),
    TO_STRING(z),
    TO_STRING(rX),
    TO_STRING(rY),
    TO_STRING(rZ),
    TO_STRING(user),
    TO_STRING(tool)
  );
ELSIF isJointNear = 0 AND jointNear <> 0 THEN
  commandOutput := CreateCommand_NineArgs(
    INVERSE_SOLUTION_CMD,
    TO_STRING(x),
    TO_STRING(y),
    TO_STRING(z),
    TO_STRING(rX),
    TO_STRING(rY),
    TO_STRING(rZ),
    TO_STRING(user),
    TO_STRING(tool),
    TO_STRING(jointNear)
  );
ELSIF isJointNear <> 0 AND jointNear = 0 THEN
    commandOutput := CreateCommand_NineArgs(
    INVERSE_SOLUTION_CMD,
    TO_STRING(x),
    TO_STRING(y),
    TO_STRING(z),
    TO_STRING(rX),
    TO_STRING(rY),
    TO_STRING(rZ),
    TO_STRING(user),
    TO_STRING(tool),
    TO_STRING(isJointNear)
  );

ELSIF isJointNear <> 0 AND jointNear <> 0 THEN
    commandOutput := CreateCommand_TenArgs(
    INVERSE_SOLUTION_CMD,
    TO_STRING(x),
    TO_STRING(y),
    TO_STRING(z),
    TO_STRING(rX),
    TO_STRING(rY),
    TO_STRING(rZ),
    TO_STRING(user),
    TO_STRING(tool),
    TO_STRING(isJointNear),
    TO_STRING(jointNear)
  );

END_IF
InverseSolution := TRUE;
END_METHOD

METHOD PalletCreate : BOOL
VAR_INPUT
	p1 : ARRAY[0..5] OF LREAL ; //Cartesian coordinates of P1, in the format {X,Y,Z,Rx,Ry,Rz}
	p2 : ARRAY[0..5] OF LREAL ; //Cartesian coordinates of P2, in the format {X,Y,Z,Rx,Ry,Rz}
	p3 : ARRAY[0..5] OF LREAL ; //Cartesian coordinates of P3, in the format {X,Y,Z,Rx,Ry,Rz}
	p4 : ARRAY[0..5] OF LREAL ; //Cartesian coordinates of P4, in the format {X,Y,Z,Rx,Ry,Rz}
	row : INT; //Rows of pallets
	col : INT; //Columns of pallets
	palletname : STRING; //Pallet name, non-repeatable
END_VAR
VAR_OUTPUT
	commandOutput : DOBOT_CMD_STRING;
END_VAR
VAR CONSTANT
  PALLET_CREATE : STRING := 'PalletCreate';
END_VAR
commandOutput := CreateCommand_SixArgs(
  arrayToString(p1),
  arrayToString(p2),
  arrayToString(p3),
  arrayToString(p4),
  TO_STRING(row),
  TO_STRING(col),
  palletname
);

PalletCreate := TRUE;
END_METHOD

METHOD PositiveSolution : BOOL
VAR_INPUT
	j1 : REAL ; //J1-axis position, unit: °
	j2 : REAL; //J2-axis position, unit: °
	j3 : REAL; //J3-axis position, unit: °
	j4 : REAL; //J4-axis position, unit: °
	j5 : REAL; //J5-axis position, unit: °
	j6 : REAL; //J6-axis position, unit: °
	user : INT; //Index of the calibrated user coordinate system
	tool : INT; //Index of the calibrated user coordinate system
END_VAR
VAR_OUTPUT
	commandOutput : DOBOT_CMD_STRING;
END_VAR
VAR CONSTANT
  POSITIVE_SOLUTION_CMD : STRING := 'PositiveSolution';
END_VAR
commandOutput := CreateCommand_EightArgs(
  POSITIVE_SOLUTION_CMD,
  TO_STRING(j1),
  TO_STRING(j2),
  TO_STRING(j3),
  TO_STRING(j4),
  TO_STRING(j5),
  TO_STRING(j6),
  TO_STRING(user),
  TO_STRING(tool)
);

PositiveSolution := TRUE;
END_METHOD

METHOD RobotMode : BOOL
VAR_OUTPUT
	commandOutput : DOBOT_CMD_STRING;
END_VAR
VAR CONSTANT
	ROBOT_MODE : STRING := 'RobotMode';
END_VAR
commandOutput := CreateCommandNoArgs(ROBOT_MODE);
RobotMode := TRUE;
END_METHOD

METHOD AnalogueInput : BOOL
VAR_INPUT
	index : INT ; //AI index
END_VAR
VAR_OUTPUT
	commandOutput : DOBOT_CMD_STRING;
END_VAR
VAR
	AI_CMD : STRING := 'AI';
END_VAR
commandOutput := CreateCommand_OneArg(AI_CMD, TO_STRING(index));
AnalogueInput := TRUE;
END_METHOD

METHOD AnalogueOutput : BOOL
VAR_INPUT
	index : INT ; //AO index
	value : REAL; //AO output
END_VAR
VAR_OUTPUT
	commandOutput : DOBOT_CMD_STRING;
END_VAR
VAR CONSTANT
  AO_CMD : STRING := 'AO';
END_VAR
commandOutput := CreateCommand_TwoArgs(AO_CMD, TO_STRING(index), TO_STRING(value));
AnalogueOutput := TRUE;
END_METHOD

METHOD AoExecute : BOOL
VAR_INPUT
	index : INT ; //AO index
	value : REAL; //AO Output
END_VAR
VAR_OUTPUT
	commandOutput : DOBOT_CMD_STRING;
END_VAR
VAR CONSTANT
  AO_EXECUTE_CMD : STRING := 'AOExecute';
END_VAR
commandOutput := CreateCommand_TwoArgs(AO_EXECUTE_CMD, TO_STRING(index), TO_STRING(value));
AoExecute := TRUE;
END_METHOD

METHOD DigitalInput : BOOL
VAR_INPUT
	index : INT ; //DI index
END_VAR
VAR_OUTPUT
	commandOutput : DOBOT_CMD_STRING;
END_VAR
VAR CONSTANT
  DI_CMD : STRING := 'DI';
END_VAR
commandOutput := CreateCommand_OneArg(DI_CMD, TO_STRING(index));
DigitalInput := TRUE;
END_METHOD

METHOD DigitalOutput : BOOL
VAR_INPUT
  index : UINT; //DO index
  status : INT; //DO status. 1: signal, 0:without signal
END_VAR
VAR
  commandBase : STRING := 'DO()';
END_VAR
VAR_OUTPUT
  commandOutput : DOBOT_CMD_STRING;
END_VAR
VAR CONSTANT
  DIGITAL_OUTPUT_CMD : STRING := 'DO';
END_VAR
commandOutput := CreateCommand_TwoArgs(DIGITAL_OUTPUT_CMD, TO_STRING(index), TO_STRING(status));
DigitalOutput := TRUE;
RETURN;
END_METHOD

METHOD DiGroup : BOOL
VAR_INPUT
	inputString : STRING ; //index1,value1,index2,value2,...,indexn,valuen
END_VAR
VAR_OUTPUT
	commandOutput : DOBOT_CMD_STRING;
END_VAR
VAR CONSTANT
  DI_GROUP_CMD : STRING := 'DIGroup';
END_VAR
commandOutput := CreateCommand_OneArg(DI_GROUP_CMD,inputString);
DiGroup := TRUE;
END_METHOD

METHOD DoExecute : BOOL
VAR_INPUT
	index : INT ; //DO index
	status : INT; //DO status. 1: signal, 0: without signal
END_VAR
VAR_OUTPUT
	commandOutput : DOBOT_CMD_STRING;
END_VAR
VAR CONSTANT
  DO_EXECUTE_CMD : STRING := 'DOExecute';
END_VAR
commandOutput := CreateCommand_TwoArgs(DO_EXECUTE_CMD, TO_STRING(index), TO_STRING(status));
DoExecute := TRUE;
END_METHOD

METHOD DoGroup : BOOL
VAR_INPUT
	inputString : STRING ; //index1,value1,index2,value2,...,indexn,valuen
END_VAR
VAR_OUTPUT
	commandOutput : DOBOT_CMD_STRING;
END_VAR
VAR CONSTANT
  DO_GROUP_CMD : STRING := 'DOGroup';
END_VAR
commandOutput := CreateCommand_OneArg(DO_GROUP_CMD, inputString);
DoGroup := TRUE;
END_METHOD

METHOD GetTerminal485 : BOOL
VAR
	commandBase : STRING := 'GetTerminal485()';
END_VAR
VAR_OUTPUT
	commandOutput : DOBOT_CMD_STRING;
END_VAR
VAR CONSTANT
  GET_TERMINAL_485_CMD : STRING := 'GetTerminal485';
END_VAR
commandOutput := CreateCommandNoArgs(GET_TERMINAL_485_CMD);
GetTerminal485 := TRUE;
END_METHOD

METHOD SetTerminal485 : BOOL
VAR_INPUT
	baudRate : DINT ; //Baud rate
END_VAR
VAR_OUTPUT
	commandOutput : DOBOT_CMD_STRING;
END_VAR
VAR CONSTANT
  SET_TERMINAL_485_CMD : STRING := 'SetTerminal485';
END_VAR
commandOutput := CreateCommand_OneArg(SET_TERMINAL_485_CMD, TO_STRING(baudRate));
SetTerminal485 := TRUE;
END_METHOD

METHOD ToolAI : BOOL
VAR_INPUT
	index : INT ; //Tool AI index
END_VAR
VAR_OUTPUT
	commandOutput : DOBOT_CMD_STRING;
END_VAR
VAR CONSTANT
  TOOL_AI_CMD : STRING := 'ToolAI';
END_VAR
commandOutput := CreateCommand_OneArg(TOOL_AI_CMD, TO_STRING(index));
ToolAI := TRUE;
END_METHOD

METHOD ToolDI : BOOL
VAR_INPUT
	index : INT ; //index
END_VAR
VAR_OUTPUT
	commandOutput : DOBOT_CMD_STRING;
END_VAR
VAR CONSTANT
  TOOL_DI_CMD : STRING := 'ToolDI';
END_VAR
commandOutput := CreateCommand_OneArg(TOOL_DI_CMD, TO_STRING(index));
ToolDI := TRUE;
END_METHOD

METHOD ToolDO : BOOL
VAR_INPUT
	index : UINT ; //Tool DO index
	status : INT; //Tool DO status. 1: signal, 0: without signal
END_VAR
VAR_OUTPUT
	commandOutput : DOBOT_CMD_STRING;
END_VAR
VAR CONSTANT
  TOOL_DO_CMD : STRING := 'ToolDO';
END_VAR
commandOutput := CreateCommand_TwoArgs(TOOL_DO_CMD, TO_STRING(index), TO_STRING(status));
ToolDO := TRUE;
END_METHOD

METHOD ToolDOExecute : BOOL
VAR_INPUT
	index : INT ; //Tool DO index
	status : INT; //Tool DO status. 1: signal, 0: without signal
END_VAR
VAR_OUTPUT
	commandOutput : DOBOT_CMD_STRING;
END_VAR
VAR CONSTANT
  TOOL_DO_EXECUTE_CMD : STRING := 'ToolDOExecute';
END_VAR
commandOutput := CreateCommand_TwoArgs(TOOL_DO_EXECUTE_CMD, TO_STRING(index), TO_STRING(status));
ToolDOExecute := TRUE;
END_METHOD

METHOD GetCoils : BOOL
VAR_INPUT
	index : INT ; //Master Index
	addr : INT; //Starting address of the coil register
	count : INT; //Number of values read from coil register, range: 1-16
END_VAR
VAR_OUTPUT
	commandOutput : DOBOT_CMD_STRING;
END_VAR
VAR CONSTANT
  GET_COILS_CMD : STRING := 'GetCoils';
END_VAR
commandOutput := CreateCommand_ThreeArgs(GET_COILS_CMD, TO_STRING(index), TO_STRING(addr), TO_STRING(count));
GetCoils := TRUE;
END_METHOD

METHOD GetHoldRegs : BOOL
VAR_INPUT
	index : INT ; //Master Index
	addr : INT; //Starting address of the holding register
	count : INT; //Number of values read from holding register, range 1-4
END_VAR
VAR_OUTPUT
	commandOutput : DOBOT_CMD_STRING;
END_VAR
VAR CONSTANT
  GET_HOLD_REGS_CMD : STRING := 'GetHoldRegs';
END_VAR
commandOutput := CreateCommand_ThreeArgs(GET_HOLD_REGS_CMD, TO_STRING(index), TO_STRING(addr), TO_STRING(count));
GetHoldRegs := TRUE;
END_METHOD

METHOD GetInBits : BOOL
VAR_INPUT
	index : INT ; //Master index
	addr : INT; //Starting address of the contact register
	count : INT; //Number of values read from contact register (discrete input), range 1-16
END_VAR
VAR_OUTPUT
	commandOutput : DOBOT_CMD_STRING;
END_VAR
VAR CONSTANT
  GET_IN_BITS_CMD : STRING := 'GetInBits';
END_VAR
commandOutput := CreateCommand_ThreeArgs(GET_IN_BITS_CMD, TO_STRING(index), TO_STRING(addr), TO_STRING(count));
GetInBits := TRUE;
END_METHOD

METHOD GetInRegs : BOOL
VAR_INPUT
	index : INT ; //Master index
	addr : INT; //Starting address of the input register
	count : INT; //number of values read from input register, range 1-4
END_VAR
VAR_OUTPUT
	commandOutput : DOBOT_CMD_STRING;
END_VAR
VAR CONSTANT
  GET_IN_REGS_CMD : STRING := 'GetInRegs';
END_VAR
commandOutput := CreateCommand_ThreeArgs(GET_IN_REGS_CMD, TO_STRING(index), TO_STRING(addr), TO_STRING(count));
GetInRegs := TRUE;
END_METHOD

METHOD ModbusClose : BOOL
VAR_INPUT
	index : INT ; //Master index
END_VAR
VAR_OUTPUT
	commandOutput : DOBOT_CMD_STRING;
END_VAR
VAR CONSTANT
  MODBUS_CLOSE_CMD : STRING := 'ModbusClose';
END_VAR
commandOutput := CreateCommand_OneArg(MODBUS_CLOSE_CMD, TO_STRING(index));
ModbusClose := TRUE;
END_METHOD

METHOD ModbusCreate : BOOL
VAR_INPUT
	ip : STRING ; //IP address of slave station. When IP is not specified, or is specified to 127.0.0.1 or 0.0.0.1, it indicates connecting to the local Modbus slave. 
	port : UINT; //Port of slave station
	slave_id : INT; //ID of slave station
	isRTU : INT; // Optional parameter. null or 0: establish ModbusTCP communicationl 1:establish ModbusRTU communication.
END_VAR
VAR_OUTPUT
	commandOutput : DOBOT_CMD_STRING;
END_VAR
VAR CONSTANT
  MODBUS_CREATE_CMD : STRING := 'ModbusCreate';
END_VAR
commandOutput := CreateCommand_FourArgs(MODBUS_CREATE_CMD, ip, TO_STRING(port), TO_STRING(slave_id), TO_STRING(isRTU));
ModbusCreate := TRUE;
END_METHOD

METHOD SetCoils : BOOL
VAR_INPUT
	index : INT ; //Master Index
	addr : INT; //Starting address of the coil register
	count : INT; //Number of values to be written to coil register, range 1-16
	valTab : STRING; //Values to be written to coil register (number of values equals to count)
END_VAR
VAR_OUTPUT
	commandOutput : DOBOT_CMD_STRING;
END_VAR
VAR CONSTANT
  SET_COILS_CMD : STRING := 'SetCoils';
END_VAR
commandOutput := CreateCommand_FourArgs(SET_COILS_CMD, TO_STRING(index), TO_STRING(addr), TO_STRING(count), valTab);
SetCoils := TRUE;
END_METHOD

METHOD SetHoldRegs : BOOL
VAR_INPUT
	index : INT ; //Master index
	addr : INT; //Starting address of the holding register
	count : INT; //Number of values to be written to the holding register, range: 1-4
	valTab : STRING; //Values to be written to the holding register (number of values equals to the count)
	valType : STRING; //Optional parameter. Data type: null or U16: 16-bit unsigned integer (two bytes, occupy one register); U32: 32-bit unsigned integer (four bytes, occupy two registers); F32: 32-bit single-precision floating-point number (four bytes, occupy two registers); F64: 64-bit double-precision floating-point number (eight bytes, occupy four registers)\
END_VAR
VAR_OUTPUT
	commandOutput : DOBOT_CMD_STRING;
END_VAR
VAR CONSTANT
  SET_HOLD_REGS_CMD : STRING := 'SetHoldRegs';
END_VAR
IF valType = '' THEN
  commandOutput := CreateCommand_FourArgs(SET_HOLD_REGS_CMD, TO_STRING(index), TO_STRING(addr), TO_STRING(count), valTab);
ELSE
  commandOutput := CreateCommand_FiveArgs(SET_HOLD_REGS_CMD, TO_STRING(index), TO_STRING(addr), TO_STRING(count), valTab, valType);
END_IF

SetHoldRegs := TRUE;
END_METHOD

METHOD Circle3 : BOOL
VAR_INPUT
	x1 : REAL ; //X-axis position of arc through point, unit: mm
	y1 : REAL ; //Y-axis position of arc through point, unit: mm
	z1 : REAL ; //Z-axis position of arc through point, unit: mm
	
	rx1 : REAL; //Rx-axis position of arc through point, unit: °
	ry1 : REAL; //Ry-axis position of arc through point, unit: °
	rz1 : REAL; //Rz-axis position of arc through point, unit: °
	
	x2 : REAL ; //X-axis position of arc through point, unit: mm
	y2 : REAL ; //Y-axis position of arc through point, unit: mm
	z2 : REAL ; //Z-axis position of arc through point, unit: mm
	
	rx2 : REAL; //Rx-axis position of arc through point, unit: °
	ry2 : REAL; //Ry-axis position of arc through point, unit: °
	rz2 : REAL; //Rz-axis position of arc through point, unit: °
	
	count : INT; //Circles of motion, range: 1-999.
END_VAR
VAR_OUTPUT
	commandOutput : DOBOT_CMD_STRING;
END_VAR
VAR CONSTANT 
  CIRCLE_3_CMD : STRING := 'Circle3';
END_VAR
commandOutput := CreateCommand_Thirteen_Args(
  CIRCLE_3_CMD,
  TO_STRING(x1), 
  TO_STRING(y1), 
  TO_STRING(z1), 
  TO_STRING(rx1),
  TO_STRING(ry1),
  TO_STRING(rz1),
  TO_STRING(x2),
  TO_STRING(y2),
  TO_STRING(z2),
  TO_STRING(rx2),
  TO_STRING(ry2),
  TO_STRING(rz2),
  TO_STRING(count)
);

Circle3 := TRUE;
  
  
  
  
  
  
  
  
  
  
  
  
  
  
  
  
  
  
  
  
  
Circle3 := TRUE;
END_METHOD

METHOD Circle3Advanced : BOOL
VAR_INPUT
	x1 : REAL ; //X-axis position of arc through point, unit: mm
	y1 : REAL ; //Y-axis position of arc through point, unit: mm
	z1 : REAL ; //Z-axis position of arc through point, unit: mm
	rx1 : REAL; //Rx-axis position of arc through point, unit: °
	ry1 : REAL; //Ry-axis position of arc through point, unit: °
	rz1 : REAL; //Rz-axis position of arc through point, unit: °
	x2 : REAL ; //X-axis position of arc through point, unit: mm
	y2 : REAL ; //Y-axis position of arc through point, unit: mm
	z2 : REAL ; //Z-axis position of arc through point, unit: mm	
	rx2 : REAL; //Rx-axis position of arc through point, unit: °
	ry2 : REAL; //Ry-axis position of arc through point, unit: °
	rz2 : REAL; //Rz-axis position of arc through point, unit: °	
	count : INT; //Circles of motion, range: 1-999.
	user : INT; //Index of the user coordinate system, range :[0,9]. The initial value of coordinate system 0 is the base coordinate system. 
	tool : INT; //Index of the tool coordinate system, range: [0,9]. The initial value of coordinate system 0 is the flange coordinate system.
END_VAR
VAR
	CIRCLE3_CMD : STRING := 'Circle3';
END_VAR
VAR_OUTPUT
	commandOutput : DOBOT_CMD_STRING;
END_VAR
commandOutput := CreateCommand_Fifteen_Args(
  CIRCLE3_CMD,
  TO_STRING(x1),
  TO_STRING(y1),
  TO_STRING(z1),
  TO_STRING(rx1),
  TO_STRING(ry1),
  TO_STRING(rz1),
  TO_STRING(x2),
  TO_STRING(y2),
  TO_STRING(z2),
  TO_STRING(rx2),
  TO_STRING(ry2),
  TO_STRING(rz2),
  TO_STRING(count),
  TO_STRING(user),
  TO_STRING(tool)
);

Circle3Advanced := TRUE;
END_METHOD

METHOD MoveJogCartesian : BOOL // TODO - add return. use enums
VAR_INPUT
	axisID : STRING ; //Jog motion axis: X, Y, Z, Rz, Rz, Ry, Rz,  Leave empty for stopping jog
	axisDirection : BOOL; //Axis Direction : True = positive direction, False = Negative direction
END_VAR
VAR
  direction : STRING;
END_VAR
VAR_OUTPUT
	commandOutput : DOBOT_CMD_STRING;
END_VAR
VAR CONSTANT
  MOVE_JOG_CMD : STRING := 'MoveJog';
END_VAR
IF axisID <> 'X' OR axisID <> 'Y' OR axisID <> 'Z' OR axisID <> 'Rx' OR axisID <> 'Ry' OR axisID <> 'Rz' THEN
  LogError('Invald axis ID');
  RETURN;
END_IF

direction := SEL(axisDirection, '-', '+');
commandOutput := CreateCommand_TwoArgs(MOVE_JOG_CMD, axisID, direction);
MoveJogCartesian := TRUE;
END_METHOD

METHOD MoveJogCartesianAdvanced : BOOL // TODO - add return. use enums
VAR_INPUT
	axisID : STRING ; //Jog motion axis:  X, Y, Z, Rz, Rz, Ry, Rz,  Leave empty for stopping jog
	axisDirection : BOOL; //Axis Direction : True = positive direction, False = Negative direction
	coordType : INT; // set to 0 to leave default
	user : INT; // set to 0 to leave default
	tool : INT; // set to 0 to leave default
END_VAR
VAR
  direction : STRING;
END_VAR
VAR_OUTPUT
	commandOutput : DOBOT_CMD_STRING;
END_VAR
VAR CONSTANT
  MOVE_JOG_CMD : STRING := 'MoveJog';
END_VAR
IF axisID <> 'X' OR axisID <> 'Y' OR axisID <> 'Z' OR axisID <> 'Rx' OR axisID <> 'Ry' OR axisID <> 'Rz' THEN
  LogError('Invald axis ID');
  RETURN;
END_IF

direction := SEL(axisDirection, '-', '+');
commandOutput := CreateCommand_FourArgs(MOVE_JOG_CMD, axisID, direction, TO_STRING(user), TO_STRING(tool));
MoveJogCartesianAdvanced := TRUE;
END_METHOD

METHOD MoveJogJointAxis : BOOL
VAR_INPUT
	axisID : UDINT ; //Jog motion axis: 1, 2, 3, 4, 5, 6,  0 for stopping jog
	axisDirection : BOOL; //Axis Direction : True = positive direction, False = Negative direction
END_VAR
VAR_OUTPUT
	commandOutput : DOBOT_CMD_STRING;
END_VAR
VAR CONSTANT
  MOVE_JOG_CMD : STRING := 'MoveJog';
END_VAR
commandOutput := CreateCommand_TwoArgs(MOVE_JOG_CMD, TO_STRING(axisID), SEL(axisDirection, '-', '+'));
MoveJogJointAxis := TRUE;
END_METHOD

METHOD MoveJogJointAxisAdvanced : BOOL
VAR_INPUT
	axisID : UDINT ; //Jog motion axis: 1, 2, 3, 4, 5, 6,  0 for stopping jog
	axisDirection : BOOL; //Axis Direction : True = positive direction, False = Negative direction
	coordType : INT; // set to 0 to leave default
	user : INT; // set to 0 to leave default
	tool : INT; // set to 0 to leave default
END_VAR
VAR
	commandBase : STRING := 'MoveJog()';
END_VAR
VAR_OUTPUT
	commandOutput : STRING;
END_VAR
IF axisID = 0 THEN
	commandOutput := INSERT(commandBase, CONCAT('J', CONCAT(UDINT_TO_STRING(axisID),'+')), len(commandBase)-1);		
ELSE
	IF axisDirection THEN
		commandOutput := INSERT(commandBase, CONCAT('J', CONCAT(UDINT_TO_STRING(axisID),'+')), len(commandBase)-1);
	ELSE 
		commandOutput := INSERT(commandBase, CONCAT('J', CONCAT(UDINT_TO_STRING(axisID),'-')), len(commandBase)-1);
	END_IF
END_IF
IF coordType <> 0 THEN
	commandOutput := INSERT(commandOutput, CONCAT(',',INT_TO_STRING(coordType)), LEN(commandOutput)-1);
ELSIF user <> 0 THEN
	commandOutput := INSERT(commandOutput, CONCAT(',User=',INT_TO_STRING(user)), len(commandOutput)-1);
ELSIF tool <> 0 THEN
	commandOutput := INSERT(commandOutput, CONCAT(',Tool=',INT_TO_STRING(tool)), len(commandOutput)-1);	
END_IF
MoveJogJointAxisAdvanced := TRUE;
RETURN;
END_METHOD

METHOD JointMovJ : BOOL
VAR_INPUT
	j1 : REAL ; //J1-axis position of the target point, unit: °
	j2 : REAL ; //J1-axis position of the target point, unit: °
	j3 : REAL ; //J1-axis position of the target point, unit: °
	j4 : REAL ; //J1-axis position of the target point, unit: °
	j5 : REAL ; //J1-axis position of the target point, unit: °
	j6 : REAL ; //J1-axis position of the target point, unit: °
END_VAR
VAR_OUTPUT
	commandOutput : DOBOT_CMD_STRING;
END_VAR
VAR CONSTANT
  JOINT_MOVE_J_CMD : STRING := 'JointMovJ';
END_VAR
commandOutput := CreateCommand_SixArgs(
  JOINT_MOVE_J_CMD,
  TO_STRING(j1),
  TO_STRING(j2),
  TO_STRING(j3),
  TO_STRING(j4),
  TO_STRING(j5),
  TO_STRING(j6)
);

JointMovJ := TRUE;
END_METHOD

METHOD JointMovJAdvanced : BOOL
VAR_INPUT
	j1 : REAL ; //J1-axis position of the target point, unit: °
	j2 : REAL ; //J1-axis position of the target point, unit: °
	j3 : REAL ; //J1-axis position of the target point, unit: °
	j4 : REAL ; //J1-axis position of the target point, unit: °
	j5 : REAL ; //J1-axis position of the target point, unit: °
	j6 : REAL ; //J1-axis position of the target point, unit: °
	speedJ : INT; //Speed ratio: [1-100]
	accJ : INT; //Acceleration ratio: [1-100]
END_VAR
VAR_OUTPUT
	commandOutput : DOBOT_CMD_STRING;
END_VAR
VAR CONSTANT
  JOINT_MOVE_J_CMD : STRING := 'JointMovJ';
END_VAR
commandOutput := CreateCommand_EightArgs(
  JOINT_MOVE_J_CMD,
  TO_STRING(j1),
  TO_STRING(j2),
  TO_STRING(j3),
  TO_STRING(j4),
  TO_STRING(j5),
  TO_STRING(j6),
  CONCAT('SpeedJ=',TO_STRING(speedJ)),
  CONCAT('AccJ=',TO_STRING(accJ))
);

JointMovJAdvanced := TRUE;
END_METHOD

METHOD MovJ : BOOL
VAR_INPUT
	x : REAL ; //X-axis position of the target point, unit: mm
	y : REAL ; //X-axis position of the target point, unit: mm
	z : REAL ; //X-axis position of the target point, unit: mm
	rX : REAL; //Rx-axis position of the target point, unit: °
	rY : REAL; //Rx-axis position of the target point, unit: °
	rZ : REAL; //Rx-axis position of the target point, unit: °
END_VAR
VAR_OUTPUT
	commandOutput : DOBOT_CMD_STRING;
END_VAR
VAR CONSTANT
  MOVE_JOINT_CMD : STRING := 'MovJ';
END_VAR
commandOutput := CreateCommand_SixArgs(
  MOVE_JOINT_CMD,
  TO_STRING(x),
  TO_STRING(y),
  TO_STRING(z),
  TO_STRING(Rx),
  TO_STRING(Ry),
  TO_STRING(Rz)
);

MovJ := TRUE;
END_METHOD

METHOD MovJAdvanced : BOOL
VAR_INPUT
	x : REAL ; //X-axis position of the target point, unit: mm
	y : REAL ; //X-axis position of the target point, unit: mm
	z : REAL ; //X-axis position of the target point, unit: mm
	rX : REAL; //Rx-axis position of the target point, unit: °
	rY : REAL; //Rx-axis position of the target point, unit: °
	rZ : REAL; //Rx-axis position of the target point, unit: °
	speedJ : INT; //Speed ratio: [1-100]
	accJ : INT; //Acceleration ratio: [1-100]
END_VAR
VAR_OUTPUT
	commandOutput : DOBOT_CMD_STRING;
END_VAR
VAR CONSTANT
  MOVE_JOINT_CMD : STRING := 'MovJ';
END_VAR
commandOutput := CreateCommand_EightArgs(
  MOVE_JOINT_CMD,
	TO_STRING(x),
	TO_STRING(y), 
	TO_STRING(z), 
	TO_STRING(rX),
	TO_STRING(rY),
	TO_STRING(rZ),
	TO_STRING(speedJ),
	TO_STRING(accJ)
);
MovJAdvanced := TRUE;
END_METHOD

METHOD MovJIO : BOOL
VAR_INPUT
	x : REAL ; //X-axis position of the target point, unit: mm
	y : REAL ; //X-axis position of the target point, unit: mm
	z : REAL ; //X-axis position of the target point, unit: mm
	rX : REAL; //Rx-axis position of the target point, unit: °
	rY : REAL; //Rx-axis position of the target point, unit: °
	rZ : REAL; //Rx-axis position of the target point, unit: °
	di : STRING; //{Mode,Distance,Index,Status}: digital output parameters, used to set the specified DO to be triggered when the robot arm moves to a specified distance or percentage. Multiple groups of parameters can be set.
END_VAR
VAR_OUTPUT
	commandOutput : DOBOT_CMD_STRING;
END_VAR
VAR CONSTANT
  MOVE_JOINT_IO : STRING := 'MovJIO';
END_VAR
commandOutput := CreateCommand_SevenArgs(
  MOVE_JOINT_IO,
  TO_STRING(x),
  TO_STRING(y),
  TO_STRING(z),
  TO_STRING(rX),
  TO_STRING(rY),
  TO_STRING(rZ),
  di
);

MovJIO := TRUE;
END_METHOD

METHOD MovJIOAdvanced : BOOL
VAR_INPUT
	x : REAL ; //X-axis position of the target point, unit: mm
	y : REAL ; //X-axis position of the target point, unit: mm
	z : REAL ; //X-axis position of the target point, unit: mm
	rX : REAL; //Rx-axis position of the target point, unit: °
	rY : REAL; //Rx-axis position of the target point, unit: °
	rZ : REAL; //Rx-axis position of the target point, unit: °
	di : STRING; //{Mode,Distance,Index,Status}: digital output parameters, used to set the specified DO to be triggered when the robot arm moves to a specified distance or percentage. Multiple groups of parameters can be set.
	speedJ : INT; //Speed ratio: [1-100]
	accJ : INT; //Acceleration ratio: [1-100]
END_VAR
VAR_OUTPUT
	commandOutput : DOBOT_CMD_STRING;
END_VAR
VAR CONSTANT
  MOVE_JOINT_IO : STRING := 'MovJIO';
END_VAR
commandOutput := CreateCommand_NineArgs(
  MOVE_JOINT_IO,
  TO_STRING(x),
  TO_STRING(y),
  TO_STRING(z),
  TO_STRING(rX),
  TO_STRING(rY),
  TO_STRING(rZ),
  di,
  TO_STRING(speedJ),
  TO_STRING(accJ)
);

MovJIOAdvanced := TRUE;
END_METHOD

METHOD MovL : BOOL
VAR_INPUT
  x : REAL; //X-axis position of the target point, unit: mm
  y : REAL; //X-axis position of the target point, unit: mm
  z : REAL; //X-axis position of the target point, unit: mm
  rX : REAL; //Rx-axis position of the target point, unit: °
  rY : REAL; //Rx-axis position of the target point, unit: °
  rZ : REAL; //Rx-axis position of the target point, unit: °
END_VAR
VAR_OUTPUT
  commandOutput : DOBOT_CMD_STRING;
END_VAR
VAR CONSTANT
  MOVE_LINEAR_CMD : STRING := 'MovL';
END_VAR
commandOutput := CreateCommand_SixArgs(
  MOVE_LINEAR_CMD,
  TO_STRING(x),
  TO_STRING(y),
  TO_STRING(z),
  TO_STRING(Rx),
  TO_STRING(Ry),
  TO_STRING(Rz)
);

MovL := TRUE;
END_METHOD

METHOD MovLAdvanced : BOOL
VAR_INPUT
	x : REAL ; //X-axis position of the target point, unit: mm
	y : REAL ; //X-axis position of the target point, unit: mm
	z : REAL ; //X-axis position of the target point, unit: mm
	rX : REAL; //Rx-axis position of the target point, unit: °
	rY : REAL; //Rx-axis position of the target point, unit: °
	rZ : REAL; //Rx-axis position of the target point, unit: °
	user : INT; //Index of the user coordinate system, range :[0,9]. The initial value of coordinate system 0 is the base coordinate system. 
	tool : INT; //Index of the tool coordinate system, range: [0,9]. The initial value of coordinate system 0 is the flange coordinate system.
	speedL : INT; //Speed ratio: [1-100]
	accL : INT; //Acceleration ratio: [1-100]
END_VAR
VAR_OUTPUT
  commandOutput : DOBOT_CMD_STRING;
END_VAR
VAR CONSTANT
  MOVE_LINEAR_CMD : STRING := 'MovL';
END_VAR
commandOutput := CreateCommand_TenArgs(
  MOVE_LINEAR_CMD,
  TO_STRING(x),
  TO_STRING(y),
  TO_STRING(z),
  TO_STRING(Rx),
  TO_STRING(Ry),
  TO_STRING(Rz),
  CONCAT('User=',TO_STRING(user)),
  CONCAT('Tool=',TO_STRING(tool)),
  CONCAT('SpeedL=',TO_STRING(speedL)),
  CONCAT('AccL=',TO_STRING(accL))
);

MovLAdvanced := TRUE;
END_METHOD

METHOD MovLIO : BOOL
VAR_INPUT
	x 			: REAL ; //X-axis position of the target point, unit: mm
	y 			: REAL ; //X-axis position of the target point, unit: mm
	z 			: REAL ; //X-axis position of the target point, unit: mm
	rX 			: REAL; //Rx-axis position of the target point, unit: °
	rY 			: REAL; //Rx-axis position of the target point, unit: °
	rZ 			: REAL; //Rx-axis position of the target point, unit: °
	di 			: STRING; //{Mode,Distance,Index,Status}: digital output parameters, used to set the specified DO to be triggered when the robot arm moves to a specified distance or percentage. Multiple groups of parameters can be set.
END_VAR
VAR_OUTPUT
	commandOutput : DOBOT_CMD_STRING;
END_VAR
VAR CONSTANT
	MOVE_LINEAR_CMD : STRING := 'MovL';
END_VAR
commandOutput := CreateCommand_SevenArgs(
  MOVE_LINEAR_CMD,
  TO_STRING(x),
  TO_STRING(y),
  TO_STRING(z),
  TO_STRING(rX),
  TO_STRING(rY),
  TO_STRING(rZ),
  di
);
MovLIO := TRUE;
END_METHOD

METHOD MovLIOAdvanced : BOOL
VAR_INPUT
  x : REAL; //X-axis position of the target point, unit: mm
  y : REAL; //X-axis position of the target point, unit: mm
  z : REAL; //X-axis position of the target point, unit: mm
  rX : REAL; //Rx-axis position of the target point, unit: °
  rY : REAL; //Rx-axis position of the target point, unit: °
  rZ : REAL; //Rx-axis position of the target point, unit: °
  di : STRING; //{Mode,Distance,Index,Status}: digital output parameters, used to set the specified DO to be triggered when the robot arm moves to a specified distance or percentage. Multiple groups of parameters can be set.
  user : INT; //Index of the user coordinate system, range :[0,9]. The initial value of coordinate system 0 is the base coordinate system. 
  tool : INT; //Index of the tool coordinate system, range: [0,9]. The initial value of coordinate system 0 is the flange coordinate system.
  speedL : INT; //Speed ratio: [1-100]
  accL : INT; //Acceleration ratio: [1-100]

END_VAR
VAR_OUTPUT
  commandOutput : DOBOT_CMD_STRING;
END_VAR
VAR CONSTANT
  MOVE_LINEAR_CMD : STRING := 'MovL';
END_VAR
commandOutput := CreateCommand_ElevenArgs(
  MOVE_LINEAR_CMD,
  TO_STRING(x),
  TO_STRING(y),
  TO_STRING(z),
  TO_STRING(rX),
  TO_STRING(rY),
  TO_STRING(rZ),
  di,
  TO_STRING(user),
  TO_STRING(tool),
  TO_STRING(speedL),
  TO_STRING(accL)
);

MovLIOAdvanced := TRUE;
END_METHOD

METHOD RelJointMovJ : BOOL
VAR_INPUT
	offset1 : REAL ; //J1-axis offset, unit: °
	offset2 : REAL ; //J2-axis offset, unit: °
	offset3 : REAL ; //J3-axis offset, unit: °
	offset4 : REAL ; //J4-axis offset, unit: °
	offset5 : REAL ; //J5-axis offset, unit: °
	offset6 : REAL ; //J6-axis offset, unit: °
END_VAR
VAR_OUTPUT
	commandOutput : DOBOT_CMD_STRING;
END_VAR
VAR CONSTANT
	REL_JOINT_MOVEJ_CMD  : STRING := 'RelJointMovJ';
END_VAR
commandOutput := CreateCommand_SixArgs(
  REL_JOINT_MOVEJ_CMD,
  TO_STRING(offset1),
  TO_STRING(offset2),
  TO_STRING(offset3),
  TO_STRING(offset4),
  TO_STRING(offset5),
  TO_STRING(offset6)
  );
RelJointMovJ := TRUE;
END_METHOD

METHOD RelJointMovJAdvanced : BOOL
VAR_INPUT
	offset1 : REAL ; //J1-axis offset, unit: °
	offset2 : REAL ; //J2-axis offset, unit: °
	offset3 : REAL ; //J3-axis offset, unit: °
	offset4 : REAL ; //J4-axis offset, unit: °
	offset5 : REAL ; //J5-axis offset, unit: °
	offset6 : REAL ; //J6-axis offset, unit: °
	
	speedJ : INT;
	accJ : INT;
END_VAR
VAR_OUTPUT
	commandOutput : DOBOT_CMD_STRING;
END_VAR
VAR CONSTANT
	REL_JOINT_MOVEJ_CMD  : STRING := 'RelJointMovJ';
END_VAR
commandOutput := CreateCommand_EightArgs(
  REL_JOINT_MOVEJ_CMD,
  TO_STRING(offset1),
  TO_STRING(offset2),
  TO_STRING(offset3),
  TO_STRING(offset4),
  TO_STRING(offset5),
  TO_STRING(offset6),
  TO_STRING(speedJ),
  TO_STRING(accJ)
);

RelJointMovJAdvanced := TRUE;
END_METHOD

METHOD RelMovJTool : BOOL
VAR_INPUT
	offsetX : REAL ; //X-axis offset, unit: mm
	offsetY : REAL ; //Y-axis offset, unit: mm
	offsetZ : REAL ; //Z-axis offset, unit: mm
	offsetRx : REAL; //Rx-axis offset, unit: °
	offsetRy : REAL; //Ry-axis offset, unit: °
	offsetRz : REAL; //Rz-axis offset, unit: °	
	tool : INT; //Select the index of the calibrated tool coordinate system
END_VAR
VAR_OUTPUT
	commandOutput : DOBOT_CMD_STRING;
END_VAR
VAR CONSTANT 
	REL_MOVE_J_TOOL_CMD : STRING := 'RelMovJTool';
END_VAR
commandOutput := CreateCommand_SevenArgs(
  REL_MOVE_J_TOOL_CMD,
  TO_STRING(offsetX),
  TO_STRING(offsetY),
  TO_STRING(offsetZ), 
  TO_STRING(offsetRx),
  TO_STRING(offsetRy),
  TO_STRING(offsetRz),
  TO_STRING(tool)
);
  
RelMovJTool := TRUE;
END_METHOD

METHOD RelMovJToolAdvanced : BOOL
VAR_INPUT
	offsetX : REAL ; //X-axis offset, unit: mm
	offsetY : REAL ; //Y-axis offset, unit: mm
	offsetZ : REAL ; //Z-axis offset, unit: mm
	offsetRx : REAL; //Rx-axis offset, unit: °
	offsetRy : REAL; //Ry-axis offset, unit: °
	offsetRz : REAL; //Rz-axis offset, unit: °
	tool : INT; //Select the index of the calibrated tool coordinate system
	speedJ : INT;
	accJ : INT;
	toolIndex : INT;
END_VAR
VAR_OUTPUT
	commandOutput : DOBOT_CMD_STRING;
END_VAR
VAR CONSTANT 
	REL_MOVE_J_TOOL_CMD : STRING := 'RelMovJTool';
END_VAR
commandOutput := CreateCommand_TenArgs(
  REL_MOVE_J_TOOL_CMD,
  TO_STRING(offsetX),
  TO_STRING(offsetY),
  TO_STRING(offsetZ),
  TO_STRING(offsetRx),
  TO_STRING(offsetRy),
  TO_STRING(offsetRz),
  TO_STRING(tool),
  TO_STRING(speedJ),
  TO_STRING(accJ),
  TO_STRING(toolIndex),
);

RelMovJToolAdvanced := TRUE;
END_METHOD

METHOD RelMovJUser : BOOL
VAR_INPUT
	offsetX : REAL ; //X-axis offset, unit: mm
	offsetY : REAL ; //Y-axis offset, unit: mm
	offsetZ : REAL ; //Z-axis offset, unit: mm	
	offsetRx : REAL; //Rx-axis offset, unit: °
	offsetRy : REAL; //Ry-axis offset, unit: °
	offsetRz : REAL; //Rz-axis offset, unit: °
	user : INT; //Select the index of the calibrated user coordinate system
END_VAR
VAR_OUTPUT
	commandOutput : DOBOT_CMD_STRING;
END_VAR
VAR CONSTANT
	REL_MOVE_J_USER_CMD : STRING := 'RelMovJUser';
END_VAR
commandOutput := CreateCommand_SevenArgs(
  REL_MOVE_J_USER_CMD,
  TO_STRING(offsetX),
  TO_STRING(offsetY),
  TO_STRING(offsetZ), 
  TO_STRING(offsetRx),
  TO_STRING(offsetRy),
  TO_STRING(offsetRz),
  TO_STRING(user)
  );
 
RelMovJUser := TRUE;
END_METHOD

METHOD RelMovJUserAdvanced : BOOL
VAR_INPUT
	offsetX : REAL ; //X-axis offset, unit: mm
	offsetY : REAL ; //Y-axis offset, unit: mm
	offsetZ : REAL ; //Z-axis offset, unit: mm
	
	offsetRx : REAL; //Rx-axis offset, unit: °
	offsetRy : REAL; //Ry-axis offset, unit: °
	offsetRz : REAL; //Rz-axis offset, unit: °
	
	User : INT; //Select the index of the calibrated tool coordinate system
	speedJ : INT;
	accJ : INT;
	userIndex : INT;
END_VAR
VAR_OUTPUT
	commandOutput : DOBOT_CMD_STRING;
END_VAR
VAR CONSTANT
	REL_MOVE_J_USER_CMD : STRING := 'RelMovJUser';
END_VAR
commandOutput := CreateCommand_TenArgs(
  REL_MOVE_J_USER_CMD,
  TO_STRING(offsetX),
  TO_STRING(offsetY),
  TO_STRING(offsetZ),
  TO_STRING(offsetRx),
  TO_STRING(offsetRy),
  TO_STRING(offsetRz),
  TO_STRING(user),
  TO_STRING(speedJ),
  TO_STRING(accJ),
  TO_STRING(userIndex),
);

RelMovJUserAdvanced := TRUE;
END_METHOD

METHOD RelMovLTool : BOOL
VAR_INPUT
	offsetX : REAL ; //X-axis offset, unit: mm
	offsetY : REAL ; //Y-axis offset, unit: mm
	offsetZ : REAL ; //Z-axis offset, unit: mm
	offsetRx : REAL; //Rx-axis offset, unit: °
	offsetRy : REAL; //Ry-axis offset, unit: °
	offsetRz : REAL; //Rz-axis offset, unit: °
	tool : INT; //Select the index of the calibrated tool coordinate system
END_VAR
VAR_OUTPUT
	commandOutput : DOBOT_CMD_STRING;
END_VAR
VAR CONSTANT
	REL_MOVE_LINEAR_USER_CMD : STRING := 'RelMovLUser';	
END_VAR
commandOutput := CreateCommand_SevenArgs(
  REL_MOVE_LINEAR_USER_CMD,
  TO_STRING(offsetX),
  TO_STRING(offsetY),
  TO_STRING(offsetZ),
  TO_STRING(offsetRx),
  TO_STRING(offsetRy),
  TO_STRING(offsetRz),
  TO_STRING(tool)
);

RelMovLTool := TRUE;
END_METHOD

METHOD RelMovLToolAdvanced : BOOL
VAR_INPUT
	offsetX : REAL ; //X-axis offset, unit: mm
	offsetY : REAL ; //Y-axis offset, unit: mm
	offsetZ : REAL ; //Z-axis offset, unit: mm
	offsetRx : REAL; //Rx-axis offset, unit: °
	offsetRy : REAL; //Ry-axis offset, unit: °
	offsetRz : REAL; //Rz-axis offset, unit: °	
	tool : INT; //Select the index of the calibrated tool coordinate system
	speedL : INT;
	accL : INT;
	userIndex : INT;
END_VAR
VAR_OUTPUT
	commandOutput : DOBOT_CMD_STRING;
END_VAR
VAR CONSTANT
	REL_MOVE_LINEAR_USER_CMD : STRING := 'RelMovLUser';	
END_VAR
commandOutput := CreateCommand_TenArgs(
  REL_MOVE_LINEAR_USER_CMD,
  TO_STRING(offsetX),
  TO_STRING(offsetY),
  TO_STRING(offsetZ),
  TO_STRING(offsetRx),
  TO_STRING(offsetRy),
  TO_STRING(offsetRz),
  TO_STRING(tool),
  TO_STRING(speedL),
  TO_STRING(accL),
  TO_STRING(userIndex),
);

RelMovLToolAdvanced := TRUE;
END_METHOD

METHOD RelMovLUser : BOOL
VAR_INPUT
	offsetX : REAL ; //X-axis offset, unit: mm
	offsetY : REAL ; //Y-axis offset, unit: mm
	offsetZ : REAL ; //Z-axis offset, unit: mm
	offsetRx : REAL; //Rx-axis offset, unit: °
	offsetRy : REAL; //Ry-axis offset, unit: °
	offsetRz : REAL; //Rz-axis offset, unit: °	
	user : INT; //Select the index of the calibrated user coordinate system
END_VAR
VAR CONSTANT
	REL_MOVE_LINEAR_USER_CMD : STRING := 'RelMovLUser';
END_VAR
VAR_OUTPUT
	commandOutput : DOBOT_CMD_STRING;
END_VAR
commandOutput := CreateCommand_SevenArgs(
  REL_MOVE_LINEAR_USER_CMD,
  TO_STRING(offsetX),
  TO_STRING(offsetY),
  TO_STRING(offsetZ),
  TO_STRING(offsetRx),
  TO_STRING(offsetRy),
  TO_STRING(offsetRz),
  TO_STRING(user)
);

RelMovLUser := TRUE;
END_METHOD

METHOD RelMovLUserAdvanced : BOOL
VAR_INPUT
	offsetX : REAL ; //X-axis offset, unit: mm
	offsetY : REAL ; //Y-axis offset, unit: mm
	offsetZ : REAL ; //Z-axis offset, unit: mm
	offsetRx : REAL; //Rx-axis offset, unit: °
	offsetRy : REAL; //Ry-axis offset, unit: °
	offsetRz : REAL; //Rz-axis offset, unit: °
	User : INT; //Select the index of the calibrated tool coordinate system
	speedL : INT;
	accL : INT;
	userIndex : INT;
END_VAR
VAR CONSTANT
	REL_MOVE_LINEAR_USER_CMD : STRING := 'RelMovLUser';
END_VAR
VAR_OUTPUT
	commandOutput : DOBOT_CMD_STRING;
END_VAR
commandOutput := CreateCommand_TenArgs(
  REL_MOVE_LINEAR_USER_CMD,
  TO_STRING(offsetX),
  TO_STRING(offsetY),
  TO_STRING(offsetZ),
  TO_STRING(offsetRx),
  TO_STRING(offsetRy),
  TO_STRING(offsetRz),
  TO_STRING(user),
  TO_STRING(speedL),
  TO_STRING(accL),
  TO_STRING(userIndex),
);

RelMovLUserAdvanced := TRUE;
END_METHOD

METHOD ServoJ : BOOL
VAR_INPUT
	j1 : REAL ; //J1-axis position of the target point, unit: °
	j2 : REAL ; //J1-axis position of the target point, unit: °
	j3 : REAL ; //J1-axis position of the target point, unit: °
	j4 : REAL ; //J1-axis position of the target point, unit: °
	j5 : REAL ; //J1-axis position of the target point, unit: °
	j6 : REAL ; //J1-axis position of the target point, unit: °
END_VAR
VAR CONSTANT
	SERVOJ_CMD : STRING := 'ServoJ';
END_VAR
VAR_OUTPUT
	commandOutput : DOBOT_CMD_STRING;
END_VAR
commandOutput := CreateCommand_SixArgs(
  SERVOJ_CMD,
  TO_STRING(j1),
  TO_STRING(j2),
  TO_STRING(j3),
  TO_STRING(j4),
  TO_STRING(j5),
  TO_STRING(j6)
);
ServoJ := TRUE;
END_METHOD

METHOD ServoJAdvanced : BOOL
VAR_INPUT
  j1 : LREAL; //J1-axis position of the target point, unit: °
  j2 : LREAL; //J1-axis position of the target point, unit: °
  j3 : LREAL; //J1-axis position of the target point, unit: °
  j4 : LREAL; //J1-axis position of the target point, unit: °
  j5 : LREAL; //J1-axis position of the target point, unit: °
  j6 : LREAL; //J1-axis position of the target point, unit: °
  t : LREAL;
  lookahead_time : LREAL;
  gain : LREAL;
END_VAR
VAR CONSTANT
  SERVOJ_CMD : STRING := 'ServoJ';
END_VAR
VAR_OUTPUT
  commandOutput : DOBOT_CMD_STRING;
END_VAR
commandOutput := CreateCommand_NineArgs(
  SERVOJ_CMD,
  TO_STRING(j1),
  TO_STRING(j2),
  TO_STRING(j3),
  TO_STRING(j4),
  TO_STRING(j5),
  TO_STRING(j6),
  TO_STRING(t),
  TO_STRING(lookahead_time),
  TO_STRING(gain)
);
ServoJAdvanced := TRUE;
END_METHOD

METHOD Arc : BOOL
VAR_INPUT
	x1 : REAL ; //X-axis position of arc through point, unit: mm
	y1 : REAL ; //Y-axis position of arc through point, unit: mm
	z1 : REAL ; //Z-axis position of arc through point, unit: mm
	
	rx1 : REAL; //Rx-axis position of arc through point, unit: °
	ry1 : REAL; //Ry-axis position of arc through point, unit: °
	rz1 : REAL; //Rz-axis position of arc through point, unit: °
	
	x2 : REAL ; //X-axis position of arc through point, unit: mm
	y2 : REAL ; //Y-axis position of arc through point, unit: mm
	z2 : REAL ; //Z-axis position of arc through point, unit: mm
	
	rx2 : REAL; //Rx-axis position of arc through point, unit: °
	ry2 : REAL; //Ry-axis position of arc through point, unit: °
	rz2 : REAL; //Rz-axis position of arc through point, unit: °
END_VAR
VAR
	commandBase : STRING := 'Arc()';
	user : INT; 
	tool : INT;
	speedL : INT;
	accL : INT;
END_VAR
VAR_OUTPUT
	commandOutput : STRING;
END_VAR
commandOutput := INSERT(commandBase, REAL_TO_STRING(x1), len(commandBase)-1);
commandOutput := INSERT(commandOutput, CONCAT(',',REAL_TO_STRING(y1)), LEN(commandOutput)-1);
commandOutput := INSERT(commandOutput, CONCAT(',',REAL_TO_STRING(z1)), LEN(commandOutput)-1);

commandOutput := INSERT(commandOutput, CONCAT(',',REAL_TO_STRING(rx1)), LEN(commandOutput)-1);
commandOutput := INSERT(commandOutput, CONCAT(',',REAL_TO_STRING(ry1)), LEN(commandOutput)-1);
commandOutput := INSERT(commandOutput, CONCAT(',',REAL_TO_STRING(rz1)), LEN(commandOutput)-1);

commandOutput := INSERT(commandOutput, CONCAT(',',REAL_TO_STRING(x2)), LEN(commandOutput)-1);
commandOutput := INSERT(commandOutput, CONCAT(',',REAL_TO_STRING(y2)), LEN(commandOutput)-1);
commandOutput := INSERT(commandOutput, CONCAT(',',REAL_TO_STRING(z2)), LEN(commandOutput)-1);

commandOutput := INSERT(commandOutput, CONCAT(',',REAL_TO_STRING(rx2)), LEN(commandOutput)-1);
commandOutput := INSERT(commandOutput, CONCAT(',',REAL_TO_STRING(ry2)), LEN(commandOutput)-1);
commandOutput := INSERT(commandOutput, CONCAT(',',REAL_TO_STRING(rz2)), LEN(commandOutput)-1);
IF user <> 0 THEN
	commandOutput := INSERT(commandOutput, CONCAT(',User=',INT_TO_STRING(user)), len(commandOutput)-1);
ELSIF tool <> 0 THEN
	commandOutput := INSERT(commandOutput, CONCAT(',Tool=',INT_TO_STRING(tool)), len(commandOutput)-1);
ELSIF speedL <> 0 THEN
	commandOutput := INSERT(commandOutput, CONCAT(',SpeedL=',INT_TO_STRING(speedL)), len(commandOutput)-1);
ELSIF accL <> 0 THEN
	commandOutput := INSERT(commandOutput, CONCAT(',AccL=',INT_TO_STRING(accL)), len(commandOutput)-1);
END_IF
Arc := TRUE;
RETURN;
END_METHOD

METHOD ServoP : BOOL
VAR_INPUT
	x : REAL ; //X-axis position of the target point, unit: mm
	y : REAL ; //X-axis position of the target point, unit: mm
	z : REAL ; //X-axis position of the target point, unit: mm
	rX : REAL; //Rx-axis position of the target point, unit: °
	rY : REAL; //Rx-axis position of the target point, unit: °
	rZ : REAL; //Rx-axis position of the target point, unit: °
END_VAR
VAR CONSTANT
	SERVO_P_CMD : STRING := 'ServoP';
END_VAR
VAR_OUTPUT
	commandOutput : DOBOT_CMD_STRING;
END_VAR
commandOutput := CreateCommand_SixArgs(
  SERVO_P_CMD,
  TO_STRING(x),
  TO_STRING(y),
  TO_STRING(z),
  TO_STRING(rX),
  TO_STRING(rY),
  TO_STRING(rZ)
);

ServoP := TRUE;
END_METHOD

METHOD StartPath : BOOL
VAR_INPUT
	traceName : STRING ; //Trajectory file name (with suffix) The trajectory file is stored in /dobot/userdata/project/process/trajectory/.
	const : INT; //Whether to play back at a constant speed. 1: play back at a constant speed, and pauses will be removed from the trajectory. 0: play back at the original speed.
	cart : INT; //The type of playback path. 1: play back as Cartesian path. 0: play back as joint path.
END_VAR
VAR CONSTANT 
	START_PATH_CMD : STRING := 'StartPath';
END_VAR
VAR_OUTPUT
	commandOutput : DOBOT_CMD_STRING;
END_VAR
commandOutput := CreateCommand_ThreeArgs(START_PATH_CMD ,traceName,TO_STRING(const),TO_STRING(cart));
StartPath := TRUE;
END_METHOD

METHOD StartTrace : BOOL
VAR_INPUT
	traceName : STRING ; //Trajectory file name (with suffix) The trajectory file is stored in /dobot/userdata/project/process/trajectory/.
END_VAR
VAR CONSTANT 
	START_TRACE_CMD : STRING := 'StartTrace';
END_VAR
VAR_OUTPUT
	commandOutput : DOBOT_CMD_STRING;
END_VAR
commandOutput := CreateCommand_OneArg(START_TRACE_CMD, traceName);
StartTrace := TRUE;
END_METHOD

METHOD Sync : BOOL
VAR CONSTANT
	SYNC_CMD : STRING := 'Sync';
END_VAR
VAR_OUTPUT
	commandOutput : DOBOT_CMD_STRING;
END_VAR
commandOutput := CreateCommandNoArgs(SYNC_CMD);
Sync := TRUE;
END_METHOD

METHOD PRIVATE CreateCommand : DOBOT_CMD_STRING // do not include parens on the 
VAR_INPUT
  baseCommand : STRING; // method call without args or parens. i.e. BrakeControl
END_VAR
VAR_IN_OUT
  args : ARRAY [*] OF STRING;
END_VAR
VAR
  arrStart, arrEnd, arrInd : DINT;
  tempOutput : T_MaxString;
END_VAR
arrStart := LOWER_BOUND(args, 1);
arrEnd := UPPER_BOUND(args, 1);

tempOutput := CONCAT(baseCommand, '('); 

FOR arrInd := arrStart TO arrEnd DO
  tempOutput := CONCAT(tempOutput, args[arrInd]);

  IF arrInd < arrEnd THEN
    tempOutput := CONCAT(tempOutput, ',');
  END_IF

END_FOR

tempOutput := CONCAT(tempOutput, ')');

CreateCommand := tempOutput;
END_METHOD

METHOD PRIVATE CreateCommand_EightArgs : DOBOT_CMD_STRING // do not include parens on the 
VAR_INPUT
  baseCommand : STRING; // method call without args or parens. i.e. BrakeControl
  arg_01 : STRING;
  arg_02 : STRING;
  arg_03 : STRING;
  arg_04 : STRING;
  arg_05 : STRING;
  arg_06 : STRING;
  arg_07 : STRING;
  arg_08 : STRING;
END_VAR
VAR
  args : ARRAY[1..8] OF STRING;
  arrStart, arrEnd, arrInd : DINT;
  tempOutput : T_MaxString;
END_VAR
args[1] := arg_01;
args[2] := arg_02;
args[3] := arg_03;
args[4] := arg_04;
args[5] := arg_05;
args[6] := arg_06;
args[7] := arg_07;
args[8] := arg_08;

CreateCommand_EightArgs := CreateCommand( baseCommand := baseCommand, args := args );
END_METHOD

METHOD PRIVATE CreateCommand_ElevenArgs : DOBOT_CMD_STRING // do not include parens on the 
VAR_INPUT
  baseCommand : STRING; // method call without args or parens. i.e. BrakeControl
  arg_01 : STRING;
  arg_02 : STRING;
  arg_03 : STRING;
  arg_04 : STRING;
  arg_05 : STRING;
  arg_06 : STRING;
  arg_07 : STRING;
  arg_08 : STRING;
  arg_09 : STRING;
  arg_10 : STRING;
  arg_11 : STRING;
END_VAR
VAR
  args : ARRAY[1..11] OF STRING;
  arrStart, arrEnd, arrInd : DINT;
  tempOutput : T_MaxString;
END_VAR
args[1] := arg_01;
args[2] := arg_02;
args[3] := arg_03;
args[4] := arg_04;
args[5] := arg_05;
args[6] := arg_06;
args[7] := arg_07;
args[8] := arg_08;
args[9] := arg_09;
args[10] := arg_10;
args[11] := arg_11;

CreateCommand_ElevenArgs := CreateCommand( baseCommand := baseCommand, args := args );
END_METHOD

METHOD PRIVATE CreateCommand_Fifteen_Args : DOBOT_CMD_STRING // do not include parens on the 
VAR_INPUT
  baseCommand : STRING; // method call without args or parens. i.e. BrakeControl
  arg_01 : STRING;
  arg_02 : STRING;
  arg_03 : STRING;
  arg_04 : STRING;
  arg_05 : STRING;
  arg_06 : STRING;
  arg_07 : STRING;
  arg_08 : STRING;
  arg_09 : STRING;
  arg_10 : STRING;
  arg_11 : STRING;
  arg_12 : STRING;
  arg_13 : STRING;
  arg_14 : STRING;
  arg_15 : STRING;
END_VAR
VAR
  args : ARRAY[1..15] OF STRING;
  arrStart, arrEnd, arrInd : DINT;
  tempOutput : T_MaxString;
END_VAR
args[1] := arg_01;
args[2] := arg_02;
args[3] := arg_03;
args[4] := arg_04;
args[5] := arg_05;
args[6] := arg_06;
args[7] := arg_07;
args[8] := arg_08;
args[9] := arg_09;
args[10] := arg_10;
args[11] := arg_11;
args[12] := arg_12;
args[13] := arg_13;
args[14] := arg_14;
args[15] := arg_15;

CreateCommand_Fifteen_Args := CreateCommand(baseCommand := baseCommand, args := args);
END_METHOD

METHOD PRIVATE CreateCommand_FiveArgs : DOBOT_CMD_STRING // do not include parens on the 
VAR_INPUT
  baseCommand : STRING; // method call without args or parens. i.e. BrakeControl
  arg_01 : STRING;
  arg_02 : STRING;
  arg_03 : STRING;
  arg_04 : STRING;
  arg_05 : STRING;
END_VAR
VAR
  args : ARRAY[1..5] OF STRING;
  arrStart, arrEnd, arrInd : DINT;
  tempOutput : T_MaxString;
END_VAR
args[1] := arg_01;
args[2] := arg_02;
args[3] := arg_03;
args[4] := arg_04;
args[5] := arg_05;

CreateCommand_FiveArgs := CreateCommand( baseCommand := baseCommand, args := args );
END_METHOD

METHOD PRIVATE CreateCommand_FourArgs : DOBOT_CMD_STRING // do not include parens on the 
VAR_INPUT
  baseCommand : STRING; // method call without args or parens. i.e. BrakeControl
  arg_01 : STRING;
  arg_02 : STRING;
  arg_03 : STRING;
  arg_04 : STRING;
END_VAR
VAR
  args : ARRAY[1..4] OF STRING;
  arrStart, arrEnd, arrInd : DINT;
  tempOutput : T_MaxString;
END_VAR
args[1] := arg_01;
args[2] := arg_02;
args[3] := arg_03;
args[4] := arg_04;

CreateCommand_FourArgs := CreateCommand( baseCommand := baseCommand, args := args );
END_METHOD

METHOD PRIVATE CreateCommand_NineArgs : DOBOT_CMD_STRING // do not include parens on the 
VAR_INPUT
  baseCommand : STRING; // method call without args or parens. i.e. BrakeControl
  arg_01 : STRING;
  arg_02 : STRING;
  arg_03 : STRING;
  arg_04 : STRING;
  arg_05 : STRING;
  arg_06 : STRING;
  arg_07 : STRING;
  arg_08 : STRING;
  arg_09 : STRING;
END_VAR
VAR
  args : ARRAY[1..9] OF STRING;
  arrStart, arrEnd, arrInd : DINT;
  tempOutput : T_MaxString;
END_VAR
args[1] := arg_01;
args[2] := arg_02;
args[3] := arg_03;
args[4] := arg_04;
args[5] := arg_05;
args[6] := arg_06;
args[7] := arg_07;
args[8] := arg_08;
args[9] := arg_09;

CreateCommand_NineArgs := CreateCommand( baseCommand := baseCommand, args := args );
END_METHOD

METHOD PRIVATE CreateCommand_OneArg : DOBOT_CMD_STRING // do not include parens on the 
VAR_INPUT
  baseCommand : STRING; // method call without args or parens. i.e. BrakeControl
  arg_01 : STRING;
END_VAR
VAR
  args : ARRAY[1..1] OF STRING;
  tempOutput : T_MaxString;
END_VAR
args[1] := arg_01;

CreateCommand_OneArg := CreateCommand(baseCommand := baseCommand, args := args);
END_METHOD

METHOD PRIVATE CreateCommand_SevenArgs : DOBOT_CMD_STRING // do not include parens on the 
VAR_INPUT
  baseCommand : STRING; // method call without args or parens. i.e. BrakeControl
  arg_01 : STRING;
  arg_02 : STRING;
  arg_03 : STRING;
  arg_04 : STRING;
  arg_05 : STRING;
  arg_06 : STRING;
  arg_07 : STRING;
END_VAR
VAR
  args : ARRAY[1..7] OF STRING;
  arrStart, arrEnd, arrInd : DINT;
  tempOutput : T_MaxString;
END_VAR
args[1] := arg_01;
args[2] := arg_02;
args[3] := arg_03;
args[4] := arg_04;
args[5] := arg_05;
args[6] := arg_06;
args[7] := arg_07;

CreateCommand_SevenArgs := CreateCommand( baseCommand := baseCommand, args := args );
END_METHOD

METHOD PRIVATE CreateCommand_SixArgs : DOBOT_CMD_STRING // do not include parens on the 
VAR_INPUT
  baseCommand : STRING; // method call without args or parens. i.e. BrakeControl
  arg_01 : STRING;
  arg_02 : STRING;
  arg_03 : STRING;
  arg_04 : STRING;
  arg_05 : STRING;
  arg_06 : STRING;
END_VAR
VAR
  args : ARRAY[1..6] OF STRING;
  arrStart, arrEnd, arrInd : DINT;
  tempOutput : T_MaxString;
END_VAR
args[1] := arg_01;
args[2] := arg_02;
args[3] := arg_03;
args[4] := arg_04;
args[5] := arg_05;
args[6] := arg_06;

CreateCommand_SixArgs := CreateCommand( baseCommand := baseCommand, args := args );
END_METHOD

METHOD PRIVATE CreateCommand_TenArgs : DOBOT_CMD_STRING // do not include parens on the 
VAR_INPUT
  baseCommand : STRING; // method call without args or parens. i.e. BrakeControl
  arg_01 : STRING;
  arg_02 : STRING;
  arg_03 : STRING;
  arg_04 : STRING;
  arg_05 : STRING;
  arg_06 : STRING;
  arg_07 : STRING;
  arg_08 : STRING;
  arg_09 : STRING;
  arg_10 : STRING;
END_VAR
VAR
  args : ARRAY[1..10] OF STRING;
  arrStart, arrEnd, arrInd : DINT;
  tempOutput : T_MaxString;
END_VAR
args[1] := arg_01;
args[2] := arg_02;
args[3] := arg_03;
args[4] := arg_04;
args[5] := arg_05;
args[6] := arg_06;
args[7] := arg_07;
args[8] := arg_08;
args[9] := arg_09;
args[10] := arg_10;

CreateCommand_TenArgs := CreateCommand( baseCommand := baseCommand, args := args );
END_METHOD

METHOD PRIVATE CreateCommand_Thirteen_Args : DOBOT_CMD_STRING // do not include parens on the 
VAR_INPUT
  baseCommand : STRING; // method call without args or parens. i.e. BrakeControl
  arg_01 : STRING;
  arg_02 : STRING;
  arg_03 : STRING;
  arg_04 : STRING;
  arg_05 : STRING;
  arg_06 : STRING;
  arg_07 : STRING;
  arg_08 : STRING;
  arg_09 : STRING;
  arg_10 : STRING;
  arg_11 : STRING;
  arg_12 : STRING;
  arg_13 : STRING;
END_VAR
VAR
  args : ARRAY[1..13] OF STRING;
  arrStart, arrEnd, arrInd : DINT;
  tempOutput : T_MaxString;
END_VAR
args[1] := arg_01;
args[2] := arg_02;
args[3] := arg_03;
args[4] := arg_04;
args[5] := arg_05;
args[6] := arg_06;
args[7] := arg_07;
args[8] := arg_08;
args[9] := arg_09;
args[10] := arg_10;
args[11] := arg_11;
args[12] := arg_12;
args[13] := arg_13;

CreateCommand_Thirteen_Args := CreateCommand(baseCommand := baseCommand, args := args);
END_METHOD

METHOD PRIVATE CreateCommand_ThreeArgs : DOBOT_CMD_STRING // do not include parens on the 
VAR_INPUT
  baseCommand : STRING; // method call without args or parens. i.e. BrakeControl
  arg_01 : STRING;
  arg_02 : STRING;
  arg_03 : STRING;
END_VAR
VAR
  args : ARRAY[1..3] OF STRING;
END_VAR
args[1] := arg_01;
args[2] := arg_02;
args[3] := arg_03;

CreateCommand_ThreeArgs := CreateCommand(baseCommand := baseCommand, args := args);
END_METHOD

METHOD PRIVATE CreateCommand_TwoArgs : DOBOT_CMD_STRING // do not include parens on the 
VAR_INPUT
  baseCommand : STRING; // method call without args or parens. i.e. BrakeControl
  arg_01 : STRING;
  arg_02 : STRING;
END_VAR
VAR
  args : ARRAY[1..2] OF STRING;
END_VAR
args[1] := arg_01;
args[2] := arg_02;

CreateCommand_TwoArgs := CreateCommand(baseCommand := baseCommand, args := args);
END_METHOD

METHOD PRIVATE CreateCommandNoArgs : DOBOT_CMD_STRING // do not include parens on the 
VAR_INPUT
  baseCommand : STRING; // method call without args or parens. i.e. BrakeControl
END_VAR
VAR
  tempOutput : T_MaxString;
END_VAR
tempOutput := CONCAT(baseCommand, '(');
tempOutput := CONCAT(tempOutput, ')');

CreateCommandNoArgs := tempOutput;
END_METHOD

METHOD PRIVATE EncapsulateWithCurlyBrax : STRING
VAR_INPUT
  item : STRING;
END_VAR
EncapsulateWithCurlyBrax := F_Concat3('{', item, '}');
END_METHOD

END_FUNCTION_BLOCK

// Helpers/arrayToString
FUNCTION arrayToString : STRING
VAR_INPUT
	cartesianArray : ARRAY[1..6] OF LREAL;
END_VAR
VAR
	i : INT;
	outputString : STRING := '{}';
END_VAR

FOR i := 1 TO 6 DO 
	outputString := INSERT(outputString, CONCAT(',',LREAL_TO_STRING(cartesianArray[i])), LEN(outputString)-1);
END_FOR

END_FUNCTION

// Commands and tasks/T_NumberCommandTaskV3
FUNCTION_BLOCK T_NumberCommandTaskV3 EXTENDS T_CommandTaskV3
VAR
  _numberResult : LREAL;
END_VAR

PROPERTY PUBLIC Result : LREAL
GET
Result := _numberResult;
END_GET
END_PROPERTY

METHOD PUBLIC SetResultValue
VAR_INPUT
  value : LREAL;
END_VAR
_numberResult := value;
END_METHOD

END_FUNCTION_BLOCK

// Helpers/ByteArrayAdvanceAndClearRemaining
FUNCTION ByteArrayAdvanceAndClearRemaining : BOOL
VAR_IN_OUT
  arrayToPass : ARRAY[*] OF BYTE;
END_VAR
VAR_INPUT
  positionToAdvanceFrom : UDINT;
END_VAR
VAR
  arrStart, arrEnd  : DINT;
  arrSize, sizeToMove : UDINT;
END_VAR

arrStart := LOWER_BOUND(arrayToPass, 1);
arrEnd := UPPER_BOUND(arrayToPass, 1);
arrSize := TO_UDINT(arrEnd - arrStart) + 1;

IF TO_DINT(positionToAdvanceFrom) > arrEnd THEN
  F_LogWarning('ByteArrayAdvanceAndClearRemaining: positionToAdvanceFrom > arrEnd.');
  ByteArrayAdvanceAndClearRemaining := FALSE;
  RETURN;
  
END_IF

sizeToMove := TO_UDINT(arrEnd) - positionToAdvanceFrom + 1;

MEMMOVE(
    destAddr := ADR(arrayToPass[arrStart]),
    srcAddr := ADR(arrayToPass[positionToAdvanceFrom]),
    n := TO_UDINT(sizeToMove)
  );

// clear data after the point moved.
MEMSET(
    destAddr := ADR(arrayToPass[arrStart + TO_DINT(sizeToMove)]),
    fillByte := 0,
    n := positionToAdvanceFrom - TO_UDINT(arrStart)
  );
  
ByteArrayAdvanceAndClearRemaining := TRUE;

END_FUNCTION

// Project Information/F_GetCompany
// This function has been automatically generated from the project information.
{attribute 'signature_flag' := '1073741824'}
{attribute 'TcGenerated'}
{attribute 'no-analysis'}
FUNCTION F_GetCompany : WSTRING
VAR_INPUT
	
END_VAR

F_GetCompany := "RoboConnect";

END_FUNCTION

// Project Information/F_GetTitle
// This function has been automatically generated from the project information.
{attribute 'signature_flag' := '1073741824'}
{attribute 'TcGenerated'}
{attribute 'no-analysis'}
FUNCTION F_GetTitle : WSTRING
VAR_INPUT
	
END_VAR

F_GetTitle := "RoboConnect.Dobot";

END_FUNCTION

// Project Information/F_GetVersion
// This function has been automatically generated from the project information.
{attribute 'signature_flag' := '1073741824'}
{attribute 'TcGenerated'}
{attribute 'no-analysis'}
FUNCTION F_GetVersion : ST_LibVersion
VAR_INPUT
	
END_VAR

F_GetVersion.iMajor := 0;
F_GetVersion.iMinor := 1;
F_GetVersion.iBuild := 0;
F_GetVersion.iRevision := 0;
F_GetVersion.sVersion := '0.1.0.0';
F_GetVersion.nFlags := 0;

END_FUNCTION

// V3_API/T_DashboardV3
FUNCTION_BLOCK T_DashboardV3 EXTENDS T_NamedBase
VAR
  connection : T_V3CommandAndFeedbackBaseClass;
  commandConstructor : T_DobotCommandConstructor;
  tempTask : RoboConnect.I_task;
END_VAR

connection();

METHOD ClearError : BOOL
VAR_OUTPUT
	task	: RoboConnect.I_Task;
END_VAR
VAR 
	commandString : DOBOT_CMD_STRING;
END_VAR
IF NOT commandConstructor.ClearError(commandOutput => commandString) THEN
	ClearError := FALSE;
  LogWarning('Failed to create command ClearError');
	RETURN;
  
END_IF

ClearError := CallRobotApi_NormalPriority(commandString, task => task);
END_METHOD

METHOD Disable : BOOL
VAR_OUTPUT
	task	: RoboConnect.I_Task;
END_VAR
VAR
	commandString : DOBOT_CMD_STRING;
END_VAR
IF NOT commandConstructor.DisableRobot(commandOutput => commandString) THEN
	Disable := FALSE;
	RETURN;
  
END_IF

Disable := CallRobotApi_NormalPriority(commandString, task => task);
END_METHOD

METHOD Enable : BOOL
VAR_OUTPUT
	task	: RoboConnect.I_Task;
END_VAR
VAR 
	commandString : DOBOT_CMD_STRING;
END_VAR
IF NOT commandConstructor.EnableRobot(commandOutput => commandString) THEN
	Enable := FALSE;
  LogWarning('Failed to create command EnableRobot');
	RETURN;
  
END_IF

Enable := CallRobotApi_NormalPriority(commandString, task => task);
END_METHOD

METHOD Halt : BOOL
VAR_OUTPUT
	task	: RoboConnect.I_Task;
END_VAR
VAR 
	commandString : DOBOT_CMD_STRING;
END_VAR
IF NOT commandConstructor.pause(commandOutput => commandString) THEN
  Halt := FALSE;
  LogWarning('Failed to create command Halt');
  RETURN;

END_IF

Halt := CallRobotApi_NormalPriority(commandString, task => task);
END_METHOD

METHOD Reset : BOOL
VAR_OUTPUT
	task	: RoboConnect.I_Task;
END_VAR
VAR
	commandString : DOBOT_CMD_STRING;
END_VAR
IF NOT commandConstructor.resetRobot(commandOutput => commandString) THEN
  Reset := FALSE;
  LogWarning('Failed to create command Reset');
  RETURN;

END_IF

Reset := CallRobotApi_NormalPriority(commandString, task => task);
END_METHOD

METHOD Stop : BOOL
VAR_OUTPUT
	task	: RoboConnect.I_Task;
END_VAR
VAR
	commandString : DOBOT_CMD_STRING;
END_VAR
IF NOT commandConstructor.emergencyStop(commandOutput => commandString) THEN
  Stop := FALSE;
  LogWarning('Failed to create command Stop');
  RETURN;

END_IF

Stop := CallRobotApi(commandString, priority := E_CommandPriority.HIGH, task => task);
END_METHOD

METHOD SetAnalogOutput : BOOL
VAR_INPUT
	Index	: UINT;
	Value	: LREAL;
END_VAR
VAR_OUTPUT
	task	: RoboConnect.I_Task;
END_VAR
VAR 
  commandString : DOBOT_CMD_STRING;
END_VAR
IF NOT commandConstructor.analogueOutput(index := TO_INT(Index), value := TO_REAL(Value), commandOutput => commandString) THEN
  SetAnalogOutput := FALSE;
  LogWarning('Failed to create command SetAnalogOutput');
  RETURN;
  
END_IF

SetAnalogOutput :=
  CallRobotApi_NormalPriority(
  commandString := commandString,
  task => task
);
END_METHOD

{warning 'add method implementation '}
METHOD SetBufferMode : BOOL
VAR_INPUT
	BufferMode	: RoboConnect.E_BufferMode;
END_VAR
VAR_OUTPUT
  task : I_Task;
END_VAR
END_METHOD

METHOD SetCarteasianAcceleration : BOOL
VAR_INPUT
	Acceleration	: LREAL;
END_VAR
VAR_OUTPUT
	task	: RoboConnect.I_Task;
END_VAR
VAR 
  commandString : DOBOT_CMD_STRING;
END_VAR
IF NOT commandConstructor.accL(acc := TO_INT(Acceleration), commandOutput => commandString) THEN
	SetCarteasianAcceleration := FALSE;
  LogWarning('Failed to create command SetCarteasianAcceleration');
	RETURN;
  
END_IF

SetCarteasianAcceleration := CallRobotApi_NormalPriority(commandString, task => task);
END_METHOD

METHOD SetCartesianDynamics : BOOL
VAR_INPUT
	XDynamics : BOOL;
	YDynamics : BOOL;
	ZDynamics : BOOL;
	 
	ADynamics : BOOL;
	BDynamics : BOOL;
	CDynamics : BOOL;
END_VAR
VAR_OUTPUT
  task : I_Task;
END_VAR
VAR
	orginalCartesianDynamics : RoboConnect.ST_CartesianPoint;
END_VAR
{warning 'add implementation SetCartesianDynamics()'}
//orginalCartesianDynamics := CartesianDynamics;
//IF XDynamics THEN
//	CartesianDynamics.x := 1;
//ELSE 
//	CartesianDynamics.x := 0;
//END_IF

//IF YDynamics THEN
//	CartesianDynamics.y := 1;
//ELSE 
//	CartesianDynamics.y := 0;
//END_IF

//IF ZDynamics THEN
//	CartesianDynamics.z := 1;
//ELSE 
//	CartesianDynamics.z := 0;
//END_IF


//IF ADynamics THEN
//	CartesianDynamics.a := 1;
//ELSE 
//	CartesianDynamics.a := 0;
//END_IF

//IF BDynamics THEN
//	CartesianDynamics.b := 1;
//ELSE 
//	CartesianDynamics.b := 0;
//END_IF

//IF CDynamics THEN
//	CartesianDynamics.c := 1;
//ELSE 
//	CartesianDynamics.c := 0;
//END_IF
//IF NOT ( 	orginalCartesianDynamics.x = CartesianDynamics.x
//		AND orginalCartesianDynamics.y = CartesianDynamics.y
//		AND orginalCartesianDynamics.Z = CartesianDynamics.z
//		AND orginalCartesianDynamics.A = CartesianDynamics.a
//		AND orginalCartesianDynamics.b = CartesianDynamics.b
//		AND orginalCartesianDynamics.c = CartesianDynamics.c) THEN 
//			SetCartesianDynamics := TRUE;
//			CartesianDynamicsInitalisation := TRUE;
//END_IF
END_METHOD

METHOD SetCartesianSpeed : BOOL
VAR_INPUT
	Speed	: LREAL;
END_VAR
VAR_OUTPUT
	task	: RoboConnect.I_Task;
END_VAR
VAR 
  commandString : DOBOT_CMD_STRING;
END_VAR
IF NOT commandConstructor.speedL(speed := LREAL_TO_INT(Speed), commandOutput => commandString) THEN
	SetCartesianSpeed := FALSE;
  LogWarning('Failed to create command SetCartesianSpeed');
	RETURN;
  
END_IF

SetCartesianSpeed := CallRobotApi_NormalPriority(commandString, task => task);
END_METHOD

METHOD SetDigitalOutput : BOOL
VAR_INPUT
	Index	: UINT;
	Value	: BOOL;
END_VAR
VAR_OUTPUT
	task	: RoboConnect.I_Task;
END_VAR
VAR 
  commandString : DOBOT_CMD_STRING;
END_VAR
IF NOT commandConstructor.digitalOutput(index := Index, status := BOOL_TO_INT(Value), commandOutput => commandString) THEN
	SetDigitalOutput := FALSE;
  LogWarning('Failed to create command SetDigitalOutput');
	RETURN;
  
END_IF

SetDigitalOutput := CallRobotApi_NormalPriority(commandString, task => task);
END_METHOD

METHOD SetJointAcceleration : BOOL
VAR_INPUT
	Acceleration	: LREAL;
END_VAR
VAR_OUTPUT
	task	: RoboConnect.I_Task;
END_VAR
VAR 
  commandString : T_Maxstring;
END_VAR
IF NOT commandConstructor.accJ(acc := LREAL_TO_INT(Acceleration), commandOutput => commandString) THEN
	SetJointAcceleration := FALSE;
  LogWarning('Failed to create command SetJointAcceleration');
	RETURN;
  
END_IF

SetJointAcceleration := CallRobotApi_NormalPriority(commandString, task => task);
END_METHOD

METHOD SetJointSpeed : BOOL
VAR_INPUT
	Speed	: LREAL;
END_VAR
VAR_OUTPUT
	task	: RoboConnect.I_Task;
END_VAR
VAR 
  commandString : DOBOT_CMD_STRING;
END_VAR
IF NOT commandConstructor.speedJ(speed := LREAL_TO_INT(Speed), commandOutput => commandString) THEN
	SetJointSpeed := FALSE;
  LogWarning('Failed to create command SetJointSpeed');
	RETURN;
  
END_IF

SetJointSpeed := CallRobotApi_NormalPriority(commandString, task => task);
END_METHOD

{warning 'add method implementation '}
METHOD SetToolAnalogOutput : BOOL
VAR_INPUT
	Index	: UINT;
	Value	: LREAL;
END_VAR
VAR_OUTPUT
	task	: RoboConnect.I_Task;
END_VAR
END_METHOD

METHOD SetToolDigitalOutput : BOOL
VAR_INPUT
	Index	: UINT;
	Value	: BOOL;
END_VAR
VAR_OUTPUT
	task	: RoboConnect.I_Task;
END_VAR
VAR 
  commandString : T_Maxstring;
END_VAR
IF NOT commandConstructor.tooldo(index := index, STatus := BOOL_TO_INT(Value), commandOutput => commandString) THEN
	SetToolDigitalOutput := FALSE;
  LogWarning('Failed to create command SetToolDigitalOutput');
	RETURN;
  
END_IF

SetToolDigitalOutput := CallRobotApi_NormalPriority(commandString, task => task);
END_METHOD

METHOD SetToolFrame : BOOL
VAR_INPUT
	Frame	: RoboConnect.ST_CartesianPoint;
END_VAR
VAR_OUTPUT
	task	: RoboConnect.I_Task;
END_VAR
VAR 
  commandString : T_Maxstring; 
  
  tableString : STRING := '{,,,,,}';
END_VAR
// TODO - better ways of doing this
tableString := INSERT(tableString, LREAL_TO_STRING(Frame.c),6);
tableString := INSERT(tableString, LREAL_TO_STRING(Frame.b),5);
tableString := INSERT(tableString, LREAL_TO_STRING(Frame.a),4);
tableString := INSERT(tableString, LREAL_TO_STRING(Frame.z),3);
tableString := INSERT(tableString, LREAL_TO_STRING(Frame.y),2);
tableString := INSERT(tableString, LREAL_TO_STRING(Frame.x),1);

IF NOT commandConstructor.setTool(index := 1, table := tableString, commandOutput => commandString) THEN
	SetToolFrame := FALSE;
  LogWarning('Failed to create command SetToolFrame');
	RETURN;
  
END_IF

SetToolFrame := CallRobotApi_NormalPriority(commandString, task => task);
END_METHOD

{warning 'add method implementation '}
METHOD SetTransitionMode : BOOL
END_METHOD

METHOD SetTransitionParameter : BOOL
VAR_INPUT
	CPratio : LREAL;
END_VAR
VAR_OUTPUT
	task	: RoboConnect.I_Task;
END_VAR
VAR 
  commandString : T_Maxstring;
END_VAR
IF CPratio > 100 OR CPratio < 0 THEN
  LogWarning(CONCAT('Invalid CPratio request: ', TO_STRING(CPratio)));
  RETURN;

END_IF

IF NOT commandConstructor.Cp(ratio := CPratio, commandOutput => commandString) THEN
  SetTransitionParameter := FALSE;
  LogWarning('Failed to create command SetTransitionParameter');
	RETURN;
  
END_IF

SetTransitionParameter := CallRobotApi_NormalPriority(commandString, task => task);
END_METHOD

